(* Beckhoff Driver *)
	FBAxisToolLeftBeckhoff: FBHW_AXIS_SINGLE_BECKHOFF;
	FBAxisToolCenterBeckhoff: FBHW_AXIS_SINGLE_BECKHOFF;
	FBAxisToolRightBeckhoff: FBHW_AXIS_SINGLE_BECKHOFF;
	FBAxisToolFeederBeckhoff: FBHW_AXIS_SINGLE_BECKHOFF;
	FBAxisGrindFeederBeckhoff: FBHW_AXIS_SINGLE_BECKHOFF;
	FBLivevalueAxisToolLeftBeckhoff: FBHW_AXIS_LIVEVALUES_BECKHOFF;
	FBLivevalueAxisToolCenterBeckhoff: FBHW_AXIS_LIVEVALUES_BECKHOFF;
	FBLivevalueAxisToolRightBeckhoff: FBHW_AXIS_LIVEVALUES_BECKHOFF;
	FBLivevalueAxisToolFeederBeckhoff: FBHW_AXIS_LIVEVALUES_BECKHOFF;
	FBLivevalueAxisGrindFeederBeckhoff: FBHW_AXIS_LIVEVALUES_BECKHOFF;
	FBToolLeftMasterSlave:FBHW_AXIS_MULTI_BECKHOFF;
	FBToolCenterMasterSlave:FBHW_AXIS_MULTI_BECKHOFF;
	FBToolRightMasterSlave:FBHW_AXIS_MULTI_BECKHOFF;
	FBToolFeederMasterSlave:FBHW_AXIS_MULTI_BECKHOFF;
	FBCylToolTension : FBHW_CYL_ANALOGCYLINDER;
(*22.12.2009: KFS {    *)
	(*FBCalcToolTensionForce:FB_CALC_TOOLTENSION_FORCE;*)
	FBCalcToolTensionForce:FB_CALC_TOOLTENSION_FORCE_NEW;
	FBCylToolLeftActive:FBHW_CYL_STANDARD;
	FBCylToolRightActive:FBHW_CYL_STANDARD;
	FBCylToolCenterActive:FBHW_CYL_STANDARD;
	FBCylToolPrismaLeftActive:FBHW_CYL_STANDARD;
	FBCylToolPrismaRightActive:FBHW_CYL_STANDARD;
(*22.12.2009: KFS }   *)

(* Pointer auf Actuatoren *)
	ptrTAxisToolLeft:POINTER TO ST_AXIS;
	ptrTAxisToolCenter:POINTER TO ST_AXIS;
	ptrTAxisToolRight:POINTER TO ST_AXIS;
	ptrTAxisToolFeeder:POINTER TO ST_AXIS;
	ptrTAxisGrindFeeder:POINTER TO ST_AXIS;
	ptrTCylToolTension:POINTER TO ST_CYLINDER;
(*22.12.2009: KFS {    *)
	ptrTCylToolLeftActive:POINTER TO ST_CYLINDER;
	ptrTCylToolRightActive:POINTER TO ST_CYLINDER;
	ptrTCylToolCenterActive:POINTER TO ST_CYLINDER;
	ptrTCylToolPrismaLeftActive:POINTER TO ST_CYLINDER;
	ptrTCylToolPrismaRightActive:POINTER TO ST_CYLINDER;
	ptrTToolFeederWorkLength:POINTER TO ST_CYLINDER;
(*22.12.2009: KFS }   *)
	RisingEdgeHWConfig:R_TRIG;
	TONTickTime: TON;
	RisingEdgeSetError:R_TRIG;
	xHardwareConfigError: BOOL;
	xTmp: BOOL;
	xMicroRodActive: BOOL;
	xBeckhoffDriveActive: BOOL;
	xCkeckAcitveMovement: BOOL;

	axInputAxisToolLeftBeckhoff : ARRAY[1..8] OF BOOL;
	axInputAxisToolCenterBeckhoff : ARRAY[1..8] OF BOOL;
	axInputAxisToolRightBeckhoff : ARRAY[1..8] OF BOOL;
	axInputAxisToolFeederBeckhoff : ARRAY[1..8] OF BOOL;
	axInputAxisGrindFeederBeckhoff : ARRAY[1..8] OF BOOL;
	ii: INT;
	xFirstRead: BOOL;
	iStepResetHardware: INT;
	TONWaitReset: TON;
	rMaxWorkLength:REAL:=27;	 (* 0mm - 270mm = 0V - 10V  --> 270mm  --> Eingabe in cm! *)
	rMeasureWorkLengthCorrection:REAL:=0.4; (*Rundungs-Korrektur in cm*)
END_VAR
(****************************************************************************************************************************************************)
(***********                                            This Functionblock manage all the machine hardware                                                           ************)
(****************************************************************************************************************************************************)
(******************************************************************************************************************************************)
(****************************				              Activation Part                                                         *****************************)
(******************************************************************************************************************************************)
IF NOT(xFirstRead) THEN
	xFirstRead:=TRUE;
	TStation.THardware.TAxisToolLeft.T_RxPdoParameter.iControlWord:=6;
	TToolLeftRxPdoPara:=TStation.THardware.TAxisToolLeft.T_RxPdoParameter;
	TStation.THardware.TAxisToolCenter.T_RxPdoParameter.iControlWord:=6;
	TToolCenterRxPdoPara:=TStation.THardware.TAxisToolCenter.T_RxPdoParameter;
	TStation.THardware.TAxisToolRight.T_RxPdoParameter.iControlWord:=6;
	TToolRightRxPdoPara:=TStation.THardware.TAxisToolRight.T_RxPdoParameter;
	TStation.THardware.TAxisToolFeeder.T_RxPdoParameter.iControlWord:=6;
	TToolFeederRxPdoPara:=TStation.THardware.TAxisToolFeeder.T_RxPdoParameter;
	TStation.THardware.TAxisGrindFeeder.T_RxPdoParameter.iControlWord:=6;
	TGrindFeederRxPdoPara:=TStation.THardware.TAxisGrindFeeder.T_RxPdoParameter;
	(*06.12.2010 KFS:	{	*)
	T_Station.xOverwriteMaxToolLength:=FALSE;
	(*06.12.2010 KFS:	}	*)
END_IF;
IF TStation.TControl.xResetHardware THEN
	CASE iStepResetHardware OF
	1:	xResetControllerToolLeft:=TRUE;
		xResetControllerToolCenter:=TRUE;
		xResetControllerToolRight:=TRUE;
		xResetControllerToolFeeder:=TRUE;
		xResetControllerGrindFeeder:=TRUE;
		TONWaitReset(IN:=FALSE);
		iStepResetHardware:=iStepResetHardware + 1;
	2:	TONWaitReset(IN:=TRUE,PT:=T#100ms);
		IF TONWaitReset.Q THEN
			xResetControllerToolLeft:=FALSE;
			xResetControllerToolCenter:=FALSE;
			xResetControllerToolRight:=FALSE;
			xResetControllerToolFeeder:=FALSE;
			xResetControllerGrindFeeder:=FALSE;
			iStepResetHardware:=iStepResetHardware + 1;
		END_IF;
	3:	TStation.THardware.TAxisToolLeft.T_RxPdoParameter.iControlWord:=0;
		TToolLeftRxPdoPara:=TStation.THardware.TAxisToolLeft.T_RxPdoParameter;
		TStation.THardware.TAxisToolCenter.T_RxPdoParameter.iControlWord:=0;
		TToolCenterRxPdoPara:=TStation.THardware.TAxisToolCenter.T_RxPdoParameter;
		TStation.THardware.TAxisToolRight.T_RxPdoParameter.iControlWord:=0;
		TToolRightRxPdoPara:=TStation.THardware.TAxisToolRight.T_RxPdoParameter;
		TStation.THardware.TAxisToolFeeder.T_RxPdoParameter.iControlWord:=0;
		TToolFeederRxPdoPara:=TStation.THardware.TAxisToolFeeder.T_RxPdoParameter;
		TStation.THardware.TAxisGrindFeeder.T_RxPdoParameter.iControlWord:=0;
		TGrindFeederRxPdoPara:=TStation.THardware.TAxisGrindFeeder.T_RxPdoParameter;
		TONWaitReset(IN:=FALSE);
		iStepResetHardware:=iStepResetHardware + 1;
	4:	TONWaitReset(IN:=TRUE,PT:=T#100ms);
		IF TONWaitReset.Q THEN
			TStation.THardware.TAxisToolLeft.T_RxPdoParameter.iControlWord:=6;
			TToolLeftRxPdoPara:=TStation.THardware.TAxisToolLeft.T_RxPdoParameter;
			TStation.THardware.TAxisToolCenter.T_RxPdoParameter.iControlWord:=6;
			TToolCenterRxPdoPara:=TStation.THardware.TAxisToolCenter.T_RxPdoParameter;
			TStation.THardware.TAxisToolRight.T_RxPdoParameter.iControlWord:=6;
			TToolRightRxPdoPara:=TStation.THardware.TAxisToolRight.T_RxPdoParameter;
			TStation.THardware.TAxisToolFeeder.T_RxPdoParameter.iControlWord:=6;
			TToolFeederRxPdoPara:=TStation.THardware.TAxisToolFeeder.T_RxPdoParameter;
			TStation.THardware.TAxisGrindFeeder.T_RxPdoParameter.iControlWord:=6;
			TGrindFeederRxPdoPara:=TStation.THardware.TAxisGrindFeeder.T_RxPdoParameter;
			TONWaitReset(IN:=FALSE);
			iStepResetHardware:=1;
			TStation.TControl.xResetHardware:=FALSE;
		END_IF;
	END_CASE;
	RETURN;
ELSE
	iStepResetHardware:=1;
END_IF;
xActiveHWStation:=TStation.TControl.xActiveHardware;
RisingEdgeHWConfig(CLK:=xHardwareConfigError);
IF RisingEdgeHWConfig.Q THEN
	TStation.TControl.diErrorNr:=0;
	TStation.TControl.xError:=FALSE;
END_IF;
IF NOT(TStation.TControl.xActiveHardware) THEN
	TStation.TControl.xHWAxesActive:=TRUE;
	xHardwareConfigError:=FALSE;
	TONTickTime(IN:=FALSE);
	RisingEdgeSetError(CLK:=FALSE);
	TStation.TControl.xActiveMovement:=FALSE;
	RETURN;
ELSE
	(* Check Hardware Configuration *)
	IF TStation.TControl.xRdy THEN
		xTmp:=	(TStation.T_MachineConfig.iConfigMachineType <> iConfigMachineType) OR
				(TStation.T_MachineConfig.iConfigAxisType <> iConfigAxisType) OR
				(TStation.T_MachineConfig.iConfigVisuNavigation <> iConfigVisuNavigation) OR
				( (TStation.T_MachineConfig.rConfigMaxToolLength <> rConfigMaxToolLength) AND NOT(T_Station.xOverwriteMaxToolLength));
		IF xTmp THEN
			IF (TStation.T_MachineConfig.iConfigMachineType <> iConfigMachineType) THEN
				TStation.TControl.diErrorNr:=7001;	(* Error-->Config Machine Type changed *)
			END_IF;
			IF (TStation.T_MachineConfig.iConfigAxisType <> iConfigAxisType) THEN
				TStation.TControl.diErrorNr:=7002;	(* Error-->Config Axis Type changed *)
			END_IF;
			IF (TStation.T_MachineConfig.iConfigVisuNavigation <> iConfigVisuNavigation) THEN
				TStation.TControl.diErrorNr:=7003;	(* Error-->Config Visu Navigation changed *)
			END_IF;
			IF (TStation.T_MachineConfig.rConfigMaxToolLength <> rConfigMaxToolLength) THEN
				TStation.TControl.diErrorNr:=7004;	(* Error-->Config Max Tool Length changed *)
			END_IF;
			RisingEdgeSetError(CLK:=TRUE);
			IF RisingEdgeSetError.Q THEN
				TStation.TControl.xError:=TRUE;
			END_IF;
			xHardwareConfigError:=TRUE;
			TStation.TControl.xHardwareConfigError:=TRUE;
		END_IF;
	END_IF;
	IF xHardwareConfigError THEN
		TStation.TControl.xActiveMovement:=FALSE;
		RETURN;
	END_IF;
	IF NOT(TStation.TControl.xHardwareConfigError) THEN
		RisingEdgeSetError(CLK:=FALSE);
	END_IF;
	(* Zuweisung der Datenstrukturen der Aktuatoren als Pointer *)
	ptrTAxisToolLeft:=ADR(TStation.THardware.TAxisToolLeft);
	ptrTAxisToolCenter:=ADR(TStation.THardware.TAxisToolCenter);
	ptrTAxisToolRight:=ADR(TStation.THardware.TAxisToolRight);
	ptrTAxisToolFeeder:=ADR(TStation.THardware.TAxisToolFeeder);
	ptrTAxisGrindFeeder:=ADR(TStation.THardware.TAxisGrindFeeder);
	ptrTCylToolTension:=ADR(TStation.THardware.TCylToolTension);
(*22.12.2009: KFS {    *)
	ptrTCylToolLeftActive:=ADR(TStation.THardware.TCylToolLeftActive);
	ptrTCylToolRightActive:=ADR(TStation.THardware.TCylToolRightActive);
	ptrTCylToolCenterActive:=ADR(TStation.THardware.TCylToolCenterActive);
	ptrTCylToolPrismaLeftActive:=ADR(TStation.THardware.TCylToolPrismaLeftActive);
	ptrTCylToolPrismaRightActive:=ADR(TStation.THardware.TCylToolPrismaRightActive);
	ptrTToolFeederWorkLength:=ADR(TStation.THardware.TToolFeederWorkLength);
(*22.12.2009: KFS }   *)
	IF (iConfigMachineType = 2) THEN
		xMicroRodActive:=TRUE;
	ELSE
		xMicroRodActive:=FALSE;
	END_IF;
	IF (iConfigAxisType = 2) THEN
		xBeckhoffDriveActive:=TRUE;
	ELSE
		xBeckhoffDriveActive:=FALSE;
	END_IF;
END_IF;
(******************************************************************************************************************************************)
(****************************				         Check if Axis Active                                                    *****************************)
(******************************************************************************************************************************************)
xTmp:= ptrTAxisToolLeft^.T_CtrleSingle.xDone AND ptrTAxisToolRight^.T_CtrleSingle.xDone AND ptrTAxisToolFeeder^.T_CtrleSingle.xDone AND ptrTAxisGrindFeeder^.T_CtrleSingle.xDone;
xTmp:=xTmp AND ((ptrTAxisToolCenter^.T_CtrleSingle.xDone AND xMicroRodActive) OR NOT(xMicroRodActive));
IF xTmp THEN
	TStation.TControl.xHWAxesActive:=FALSE;
ELSE
	TStation.TControl.xHWAxesActive:=TRUE;
END_IF;
(******************************************************************************************************************************************)
(****************************	                        Check if Axis and Cylinder are Active                               *****************************)
(******************************************************************************************************************************************)
xCkeckAcitveMovement:=	(NOT(ptrTAxisToolLeft^.T_CtrleSingle.xDone) AND NOT(ptrTAxisToolLeft^.T_CtrleSingle.xErr)) OR
						(NOT(ptrTAxisToolRight^.T_CtrleSingle.xDone) AND NOT(ptrTAxisToolRight^.T_CtrleSingle.xErr)) OR
						(NOT(ptrTAxisToolFeeder^.T_CtrleSingle.xDone) AND NOT(ptrTAxisToolFeeder^.T_CtrleSingle.xErr)) OR
						(NOT(ptrTAxisGrindFeeder^.T_CtrleSingle.xDone) AND NOT(ptrTAxisGrindFeeder^.T_CtrleSingle.xErr)) OR
						(NOT(ptrTAxisToolCenter^.T_CtrleSingle.xDone) AND NOT(ptrTAxisToolCenter^.T_CtrleSingle.xErr) AND xMicroRodActive) OR
(*22.12.2009: KFS {    *)		(NOT(ptrTCylToolLeftActive^.T_CtrleCyl.xDone) AND NOT(ptrTCylToolLeftActive^.T_CtrleCyl.xErr) AND xMicroRodActive) OR
						(NOT(ptrTCylToolRightActive^.T_CtrleCyl.xDone) AND NOT(ptrTCylToolRightActive^.T_CtrleCyl.xErr) AND xMicroRodActive) OR
						(NOT(ptrTCylToolCenterActive^.T_CtrleCyl.xDone) AND NOT(ptrTCylToolCenterActive^.T_CtrleCyl.xErr) AND xMicroRodActive) OR
						(NOT(ptrTCylToolPrismaLeftActive^.T_CtrleCyl.xDone) AND NOT(ptrTCylToolPrismaLeftActive^.T_CtrleCyl.xErr) AND xMicroRodActive) OR
						(NOT(ptrTCylToolPrismaRightActive^.T_CtrleCyl.xDone) AND NOT(ptrTCylToolPrismaRightActive^.T_CtrleCyl.xErr) AND xMicroRodActive) OR	(*22.12.2009: KFS }   *)
						(NOT(ptrTCylToolTension^.T_CtrleCyl.xDone) AND NOT(ptrTCylToolTension^.T_CtrleCyl.xErr));
IF NOT(xCkeckAcitveMovement) THEN
	IF NOT(ptrTAxisToolLeft^.T_CtrleSingle.xNotMoving) AND ptrTAxisToolLeft^.T_CtrleSingle.xDone AND NOT(ptrTAxisToolLeft^.T_CtrleSingle.xErr) THEN
		xCkeckAcitveMovement:=TRUE;
	END_IF;
	IF NOT(ptrTAxisToolRight^.T_CtrleSingle.xNotMoving) AND ptrTAxisToolRight^.T_CtrleSingle.xDone AND NOT(ptrTAxisToolRight^.T_CtrleSingle.xErr) THEN
		xCkeckAcitveMovement:=TRUE;
	END_IF;
	IF NOT(ptrTAxisToolFeeder^.T_CtrleSingle.xNotMoving) AND ptrTAxisToolFeeder^.T_CtrleSingle.xDone AND NOT(ptrTAxisToolFeeder^.T_CtrleSingle.xErr) THEN
		xCkeckAcitveMovement:=TRUE;
	END_IF;
	IF NOT(ptrTAxisGrindFeeder^.T_CtrleSingle.xNotMoving) AND ptrTAxisGrindFeeder^.T_CtrleSingle.xDone AND NOT(ptrTAxisGrindFeeder^.T_CtrleSingle.xErr) THEN
		xCkeckAcitveMovement:=TRUE;
	END_IF;
	IF NOT(ptrTAxisToolCenter^.T_CtrleSingle.xNotMoving) AND ptrTAxisToolCenter^.T_CtrleSingle.xDone AND NOT(ptrTAxisToolCenter^.T_CtrleSingle.xErr) AND xMicroRodActive THEN
		xCkeckAcitveMovement:=TRUE;
	END_IF;
END_IF;
TStation.TControl.xActiveMovement:=xCkeckAcitveMovement;
IF NOT(xBeckhoffDriveActive) THEN
	(******************************************************************************************************************************************)
	(****************************				   Axis ToolLeft PDO Parameter                                      *****************************)
	(******************************************************************************************************************************************)
	TToolLeftRxPdoPara:=ptrTAxisToolLeft^.T_RxPdoParameter;
	ptrTAxisToolLeft^.T_TxPdoParameter:=TToolLeftTxPdoPara;
	(******************************************************************************************************************************************)
	(****************************				         Axis ToolLeft Live Values                                        *****************************)
	(******************************************************************************************************************************************)
	FBLivevalueAxisToolLeftEcostep(	iTypAxis:=1,
									rPrismaFactor:=0,
									xMicroRodActive:=xMicroRodActive,
									T_Axis:= ptrTAxisToolLeft^);
	(******************************************************************************************************************************************)
	(****************************				         Axis ToolLeft Motion                                                  *****************************)
	(******************************************************************************************************************************************)
	FBAxisToolLeftEcostep(	xCircuitPowerOn:= T_TwinSafeOut.QxContactor_K3 AND T_TwinSafeOut.QxContactor_K4,
							rPrismaFactor:=0,
							T_Axis:= ptrTAxisToolLeft^,
							T_HDD:= T_HDD);
	xResetControllerToolLeft:=FBAxisToolLeftEcostep.xResetController;
	xSetEnableAxisToolLeft:=FBAxisToolLeftEcostep.xSetEnableAxis;
	IF xMicroRodActive THEN
		(******************************************************************************************************************************************)
		(****************************		     	      Axis ToolCenter PDO Parameter                                      *****************************)
		(******************************************************************************************************************************************)
		TToolCenterRxPdoPara:=ptrTAxisToolCenter^.T_RxPdoParameter;
		ptrTAxisToolCenter^.T_TxPdoParameter:=TToolCenterTxPdoPara;
		(******************************************************************************************************************************************)
		(****************************				      Axis ToolCenter Live Values                                     *****************************)
		(******************************************************************************************************************************************)
		FBLivevalueAxisToolCenterEcostep(	iTypAxis:=2,
										rPrismaFactor:=0,
										xMicroRodActive:=xMicroRodActive,
										T_Axis:= ptrTAxisToolCenter^);
		(******************************************************************************************************************************************)
		(****************************				      Axis ToolCenter Motion                                               *****************************)
		(******************************************************************************************************************************************)
		FBAxisToolCenterEcostep(	xCircuitPowerOn:= T_TwinSafeOut.QxContactor_K3 AND T_TwinSafeOut.QxContactor_K4,
								rPrismaFactor:=0,
								T_Axis:= ptrTAxisToolCenter^,
								T_HDD:= T_HDD);
		xResetControllerToolCenter:=FBAxisToolCenterEcostep.xResetController;
		xSetEnableAxisToolCenter:=FBAxisToolCenterEcostep.xSetEnableAxis;
	ELSE
		xResetControllerToolCenter:=FALSE;
		xSetEnableAxisToolCenter:=FALSE;
	END_IF;
	(******************************************************************************************************************************************)
	(****************************			         Axis ToolRight PDO Parameter                                      *****************************)
	(******************************************************************************************************************************************)
	TToolRightRxPdoPara:=ptrTAxisToolRight^.T_RxPdoParameter;
	ptrTAxisToolRight^.T_TxPdoParameter:=TToolRightTxPdoPara;
	(******************************************************************************************************************************************)
	(****************************				        Axis ToolRight Live Values                                      *****************************)
	(******************************************************************************************************************************************)
	FBLivevalueAxisToolRightEcostep(	iTypAxis:=3,
									rPrismaFactor:=0,
									xMicroRodActive:=xMicroRodActive,
									T_Axis:= ptrTAxisToolRight^);
	(******************************************************************************************************************************************)
	(****************************				         Axis ToolRight Motion                                               *****************************)
	(******************************************************************************************************************************************)
	FBAxisToolRightEcostep(	xCircuitPowerOn:= T_TwinSafeOut.QxContactor_K3 AND T_TwinSafeOut.QxContactor_K4,
							rPrismaFactor:=0,
							T_Axis:= ptrTAxisToolRight^,
							T_HDD:= T_HDD);
	xResetControllerToolRight:=FBAxisToolRightEcostep.xResetController;
	xSetEnableAxisToolRight:=FBAxisToolRightEcostep.xSetEnableAxis;
	(******************************************************************************************************************************************)
	(****************************			      Axis ToolFeeder PDO Parameter                                    *****************************)
	(******************************************************************************************************************************************)
	TToolFeederRxPdoPara:=ptrTAxisToolFeeder^.T_RxPdoParameter;
	ptrTAxisToolFeeder^.T_TxPdoParameter:=TToolFeederTxPdoPara;
	(******************************************************************************************************************************************)
	(****************************				    Axis ToolFeeder Live Values                                     *****************************)
	(******************************************************************************************************************************************)
	FBLivevalueAxisToolFeederEcostep(	iTypAxis:=4,
										rPrismaFactor:=0,
										xMicroRodActive:=xMicroRodActive,
										T_Axis:= ptrTAxisToolFeeder^);
	(******************************************************************************************************************************************)
	(****************************				      Axis ToolFeeder Motion                                             *****************************)
	(******************************************************************************************************************************************)
	FBAxisToolFeederEcostep(	xCircuitPowerOn:= T_TwinSafeOut.QxContactor_K3 AND T_TwinSafeOut.QxContactor_K4,
								rPrismaFactor:=0,
								T_Axis:= ptrTAxisToolFeeder^,
								T_HDD:= T_HDD);
	xResetControllerToolFeeder:=FBAxisToolFeederEcostep.xResetController;
	xSetEnableAxisToolFeeder:=FBAxisToolFeederEcostep.xSetEnableAxis;
	(******************************************************************************************************************************************)
	(****************************			          Axis GrindFeeder PDO Parameter                               *****************************)
	(******************************************************************************************************************************************)
	TGrindFeederRxPdoPara:=ptrTAxisGrindFeeder^.T_RxPdoParameter;
	ptrTAxisGrindFeeder^.T_TxPdoParameter:=TGrindFeederTxPdoPara;
	(******************************************************************************************************************************************)
	(****************************				     Axis GrindFeeder Live Values                                   *****************************)
	(******************************************************************************************************************************************)
	FBLivevalueAxisGrindFeederEcostep(	iTypAxis:=5,
										rPrismaFactor:=rPrismaFactor,
										xMicroRodActive:=xMicroRodActive,
										T_Axis:= ptrTAxisGrindFeeder^);
	(******************************************************************************************************************************************)
	(****************************		           	      Axis GrindFeeder Motion                                            *****************************)
	(******************************************************************************************************************************************)
	FBAxisGrindFeederEcostep(	xCircuitPowerOn:= T_TwinSafeOut.QxContactor_K3 AND T_TwinSafeOut.QxContactor_K4,
								rPrismaFactor:=rPrismaFactor,
								T_Axis:= ptrTAxisGrindFeeder^,
								T_HDD:= T_HDD);
	xResetControllerGrindFeeder:=FBAxisGrindFeederEcostep.xResetController;
	xSetEnableAxisGrindFeeder:=FBAxisGrindFeederEcostep.xSetEnableAxis;
END_IF;
IF xBeckhoffDriveActive THEN
	(******************************************************************************************************************************************)
	(****************************				         Axis ToolLeft Live Values                                        *****************************)
	(******************************************************************************************************************************************)
	FOR ii:=1 TO 8 DO
		axInputAxisToolLeftBeckhoff[ii]:=axInputAxisBeckhoff[1,ii];
	END_FOR
	FBLivevalueAxisToolLeftBeckhoff(	uiActualTorque:=auiActualAxisTorqueBeckhoff[1],
									arxDigitalInput:=axInputAxisToolLeftBeckhoff,
									T_AXIS:=ptrTAxisToolLeft^,
									T_AXISRefIn:=stToolLeftRefIn);

	(******************************************************************************************************************************************)
	(****************************				         Axis ToolLeft Motion                                                  *****************************)
	(******************************************************************************************************************************************)
	FBAxisToolLeftBeckhoff(	xHWLimitPos:= FALSE,
							xHWLimitNeg:= FALSE,
							xRefHoming:= FALSE,
							T_Axis:= ptrTAxisToolLeft^,
							T_AxisRefIn:= stToolLeftRefIn,
							T_AxisRefOut:= stToolLeftRefOut,
							T_HDD:= T_HDD);

	(******************************************************************************************************************************************)
	(****************************				            Axis ToolLeft Mulit                                                    *****************************)
	(******************************************************************************************************************************************)
	IF xMicroRodActive THEN
		FBToolLeftMasterSlave(	T_AxisMaster:=ptrTAxisToolLeft^ ,
								T_AxisSlave:= ptrTAxisToolCenter^,
								T_AxisMasterRefIn:= stToolLeftRefIn,
								T_AxisSlaveRefIn:= stToolCenterRefIn);
	ELSE
		FBToolLeftMasterSlave(	T_AxisMaster:=ptrTAxisToolLeft^ ,
								T_AxisSlave:= ptrTAxisToolRight^,
								T_AxisMasterRefIn:= stToolLeftRefIn,
								T_AxisSlaveRefIn:= stToolRightRefIn);
	END_IF;

	IF xMicroRodActive THEN
		(******************************************************************************************************************************************)
		(****************************				      Axis ToolCenter Live Values                                     *****************************)
		(******************************************************************************************************************************************)
		FOR ii:=1 TO 8 DO
			axInputAxisToolCenterBeckhoff[ii]:=axInputAxisBeckhoff[2,ii];
		END_FOR
		FBLivevalueAxisToolCenterBeckhoff(	uiActualTorque:=auiActualAxisTorqueBeckhoff[2],
										arxDigitalInput:=axInputAxisToolCenterBeckhoff,
										T_AXIS:=ptrTAxisToolCenter^,
										T_AXISRefIn:=stToolCenterRefIn);

		(******************************************************************************************************************************************)
		(****************************				      Axis ToolCenter Motion                                               *****************************)
		(******************************************************************************************************************************************)
		FBAxisToolCenterBeckhoff(	xHWLimitPos:= FALSE,
								xHWLimitNeg:= FALSE,
								xRefHoming:= FALSE,
								T_Axis:= ptrTAxisToolCenter^,
								T_AxisRefIn:= stToolCenterRefIn,
								T_AxisRefOut:= stToolCenterRefOut,
								T_HDD:= T_HDD);

		(******************************************************************************************************************************************)
		(****************************				        Axis ToolCenter Mulit                                                 *****************************)
		(******************************************************************************************************************************************)
		FBToolCenterMasterSlave(	T_AxisMaster:=ptrTAxisToolCenter^ ,
								T_AxisSlave:= ptrTAxisToolRight^,
								T_AxisMasterRefIn:= stToolCenterRefIn,
								T_AxisSlaveRefIn:= stToolRightRefIn);
	END_IF;

	(******************************************************************************************************************************************)
	(****************************				        Axis ToolRight Live Values                                      *****************************)
	(******************************************************************************************************************************************)
	FOR ii:=1 TO 8 DO
		axInputAxisToolRightBeckhoff[ii]:=axInputAxisBeckhoff[3,ii];
	END_FOR
	FBLivevalueAxisToolRightBeckhoff(	uiActualTorque:=auiActualAxisTorqueBeckhoff[3],
									arxDigitalInput:=axInputAxisToolRightBeckhoff,
									T_AXIS:=ptrTAxisToolRight^,
									T_AXISRefIn:=stToolRightRefIn);

	(******************************************************************************************************************************************)
	(****************************				         Axis ToolRight Motion                                               *****************************)
	(******************************************************************************************************************************************)
	FBAxisToolRightBeckhoff(	xHWLimitPos:= FALSE,
							xHWLimitNeg:= FALSE,
							xRefHoming:= FALSE,
							T_Axis:= ptrTAxisToolRight^,
							T_AxisRefIn:= stToolRightRefIn,
							T_AxisRefOut:= stToolRightRefOut,
							T_HDD:= T_HDD);

	(******************************************************************************************************************************************)
	(****************************				            Axis ToolRight Mulit                                                *****************************)
	(******************************************************************************************************************************************)
	FBToolRightMasterSlave(	T_AxisMaster:=ptrTAxisToolRight^ ,
							T_AxisSlave:= ptrTAxisToolFeeder^,
							T_AxisMasterRefIn:= stToolRightRefIn,
							T_AxisSlaveRefIn:= stToolFeederRefIn);

	(******************************************************************************************************************************************)
	(****************************				    Axis ToolFeeder Live Values                                     *****************************)
	(******************************************************************************************************************************************)
	FOR ii:=1 TO 8 DO
		axInputAxisToolFeederBeckhoff[ii]:=axInputAxisBeckhoff[4,ii];
	END_FOR
	FBLivevalueAxisToolFeederBeckhoff(	uiActualTorque:=auiActualAxisTorqueBeckhoff[4],
										arxDigitalInput:=axInputAxisToolFeederBeckhoff,
										T_AXIS:=ptrTAxisToolFeeder^,
										T_AXISRefIn:=stToolFeederRefIn);

	(******************************************************************************************************************************************)
	(****************************				      Axis ToolFeeder Motion                                             *****************************)
	(******************************************************************************************************************************************)
	FBAxisToolFeederBeckhoff(	xHWLimitPos:= FALSE,
								xHWLimitNeg:= FALSE,
								xRefHoming:= FALSE,
								T_Axis:= ptrTAxisToolFeeder^,
								T_AxisRefIn:= stToolFeederRefIn,
								T_AxisRefOut:= stToolFeederRefOut,
								T_HDD:= T_HDD);

	(******************************************************************************************************************************************)
	(****************************				            Axis ToolFeeder Mulit                                            *****************************)
	(******************************************************************************************************************************************)
	FBToolFeederMasterSlave(T_AxisMaster:=ptrTAxisToolFeeder^ ,
							T_AxisSlave:= ptrTAxisGrindFeeder^,
							T_AxisMasterRefIn:= stToolFeederRefIn,
							T_AxisSlaveRefIn:= stGrindFeederRefIn);

	(******************************************************************************************************************************************)
	(****************************				     Axis GrindFeeder Live Values                                   *****************************)
	(******************************************************************************************************************************************)
	FOR ii:=1 TO 8 DO
		axInputAxisGrindFeederBeckhoff[ii]:=axInputAxisBeckhoff[5,ii];
	END_FOR
	FBLivevalueAxisGrindFeederBeckhoff(	uiActualTorque:=auiActualAxisTorqueBeckhoff[5],
										arxDigitalInput:=axInputAxisGrindFeederBeckhoff,
										T_AXIS:=ptrTAxisGrindFeeder^,
										T_AXISRefIn:=stGrindFeederRefIn);

	(******************************************************************************************************************************************)
	(****************************		           	      Axis GrindFeeder Motion                                            *****************************)
	(******************************************************************************************************************************************)
	FBAxisGrindFeederBeckhoff(	xHWLimitPos:= FALSE,
								xHWLimitNeg:= FALSE,
								xRefHoming:= FALSE,
								T_Axis:= ptrTAxisGrindFeeder^,
								T_AxisRefIn:= stGrindFeederRefIn,
								T_AxisRefOut:= stGrindFeederRefOut,
								T_HDD:= T_HDD);

	(******************************************************************************************************************************************)
	(****************************				           Axis GrindFeeder Mulit                                            *****************************)
	(******************************************************************************************************************************************)
	(* No Slave Axis for Axis GrindFeeder *)
END_IF;

(******************************************************************************************************************************************)
(****************************		                       Cylinder für  ToolTension                                             *****************************)
(******************************************************************************************************************************************)
FBCalcToolTensionForce(	rForcePistonIn:= ptrTCylToolTension^.T_CtrleCyl.T_AnalogCylinder.rForceIn,
						rPistonDiameterD1:= T_ParamToolTensionSystem.rPistonDiameterTT,
						rPistonDiameterD2:= T_ParamToolTensionSystem.rPistonDiameterTT2,
						rMaxAirpressure:= T_ParamToolTensionSystem.rAirPressureTT,
						rFactorForce:= T_ParamToolTensionSystem.rFactorForce);
T_ParamToolTensionSystem.rMaxForceTT:=FBCalcToolTensionForce.rSetMaxForce;
ptrTCylToolTension^.T_CtrleCyl.T_AnalogCylinder.iAnalogIN:=FBCalcToolTensionForce.iAnalogOutput;
ptrTCylToolTension^.T_CtrleCyl.T_AnalogCylinder.rForceOut:=FBCalcToolTensionForce.rForcePistonOut;
FBCylToolTension(	xCtrlePosOn:=xSensorToolTension,
					xCtrlePosOff:=FALSE,
					iAnalogIn:= ptrTCylToolTension^.T_CtrleCyl.T_AnalogCylinder.iAnalogIN,
					T_Cylinder:= ptrTCylToolTension^);
iCylOutAnaToolTension:=FBCylToolTension.iAnalogOut;
ptrTCylToolTension^.T_CtrleCyl.T_AnalogCylinder.iAnalogOut:=FBCylToolTension.iAnalogOut;
xCylOutToolTension:=FBCylToolTension.xCylinder;
IF xMicroRodActive THEN
	(* control lamp button for the Cylinder ToolTension *)
	xCtrlLampToolTensionButton:=FBCylToolTension.xCylinder;
END_IF
(******************************************************************************************************************************************)
IF xMicroRodActive THEN
	(******************************************************************************************************************************************)
	(****************************		                       Cylinder für  ToolLeftActive                                          *****************************)
	(******************************************************************************************************************************************)
	FBCylToolLeftActive(		xCtrlePosOn:= FALSE,
							xCtrlePosOff:= FALSE,
							T_Cylinder:= ptrTCylToolLeftActive^);
	xCylOutToolLeftActive:= FBCylToolLeftActive.xCylinder;
	(* control lamp button for the Cylinder ToolLeft *)
	xCtrlLampToolLeftButton:= FBCylToolLeftActive.xCylinder;
	(******************************************************************************************************************************************)
	(****************************		                       Cylinder für  ToolRightActive                                       *****************************)
	(******************************************************************************************************************************************)
	FBCylToolRightActive(		xCtrlePosOn:= FALSE,
							xCtrlePosOff:= FALSE,
							T_Cylinder:= ptrTCylToolRightActive^);
	xCylOutToolRightActive:= FBCylToolRightActive.xCylinder;
	(* control lamp button for the Cylinder ToolRight*)
	xCtrlLampToolRightButton:= FBCylToolRightActive.xCylinder;
	(******************************************************************************************************************************************)
	(****************************		                       Cylinder für  ToolCenterActive                                       *****************************)
	(******************************************************************************************************************************************)
	FBCylToolCenterActive(	xCtrlePosOn:= FALSE,
							xCtrlePosOff:= FALSE,
							T_Cylinder:= ptrTCylToolCenterActive^);
	xCylOutToolCenterActive:= FBCylToolCenterActive.xCylinder;
	(* control lamp button for the Cylinder ToolCenter *)
	xCtrlLampToolCenterButton:= FBCylToolCenterActive.xCylinder;
	(******************************************************************************************************************************************)
	(****************************		                       Cylinder für  ToolPrismaLeftActive                            *****************************)
	(******************************************************************************************************************************************)
	FBCylToolPrismaLeftActive(	xCtrlePosOn:= FALSE,
								xCtrlePosOff:= FALSE,
								T_Cylinder:= ptrTCylToolPrismaLeftActive^);
	xCylOutToolPrismaLeftActive:= FBCylToolPrismaLeftActive.xCylinder;
	(* control lamp button for the Cylinder ToolPrismaLeft *)
	xCtrlLampToolPrismaLeftButton:= FBCylToolPrismaLeftActive.xCylinder;
	(******************************************************************************************************************************************)
	(****************************		                       Cylinder für  ToolPrismaRightActive                         *****************************)
	(******************************************************************************************************************************************)
	FBCylToolPrismaRightActive(	xCtrlePosOn:= FALSE,
								xCtrlePosOff:= FALSE,
								T_Cylinder:= ptrTCylToolPrismaRightActive^);
	xCylOutToolPrismaRightActive:= FBCylToolPrismaRightActive.xCylinder;
	(* control lamp button for the Cylinder ToolPrismaRight *)
	xCtrlLampToolPrismaRightButton:= FBCylToolPrismaRightActive.xCylinder;
	(************************************************************************************************************************************************************)
	(****************************		              Calculation for the ToolFeederWorkLength                    ***********************************************)
	(************************************************************************************************************************************************************)
	ptrTToolFeederWorkLength^.T_CtrleCyl.T_Analog.rLengthIn:=((rMaxWorkLength/32767) * INT_TO_REAL(iAToolFeederWorkLength)) - rMeasureWorkLengthCorrection;
	(************************************************************************************************************************************************************)
END_IF;
(******************************************************************************************************************************************)
(****************************		                              Reset Control Flags                                                *****************************)
(******************************************************************************************************************************************)
ptrTAxisToolLeft^.T_CtrleSingle.xExecute:=FALSE;
ptrTAxisToolLeft^.T_CtrleSingle.xReset:=FALSE;
ptrTAxisToolCenter^.T_CtrleSingle.xExecute:=FALSE;
ptrTAxisToolCenter^.T_CtrleSingle.xReset:=FALSE;
ptrTAxisToolRight^.T_CtrleSingle.xExecute:=FALSE;
ptrTAxisToolRight^.T_CtrleSingle.xReset:=FALSE;
ptrTAxisToolFeeder^.T_CtrleSingle.xExecute:=FALSE;
ptrTAxisToolFeeder^.T_CtrleSingle.xReset:=FALSE;
ptrTAxisGrindFeeder^.T_CtrleSingle.xExecute:=FALSE;
ptrTAxisGrindFeeder^.T_CtrleSingle.xReset:=FALSE;
ptrTCylToolTension^.T_CtrleCyl.xReset:=FALSE;
ptrTCylToolTension^.T_CtrleCyl.xExecute:=FALSE;
ptrTCylToolLeftActive^.T_CtrleCyl.xReset:=FALSE;
ptrTCylToolLeftActive^.T_CtrleCyl.xExecute:=FALSE;
ptrTCylToolRightActive^.T_CtrleCyl.xReset:=FALSE;
ptrTCylToolRightActive^.T_CtrleCyl.xExecute:=FALSE;
ptrTCylToolCenterActive^.T_CtrleCyl.xReset:=FALSE;
ptrTCylToolCenterActive^.T_CtrleCyl.xExecute:=FALSE;
ptrTCylToolPrismaLeftActive^.T_CtrleCyl.xReset:=FALSE;
ptrTCylToolPrismaLeftActive^.T_CtrleCyl.xExecute:=FALSE;
ptrTCylToolPrismaRightActive^.T_CtrleCyl.xReset:=FALSE;
ptrTCylToolPrismaRightActive^.T_CtrleCyl.xExecute:=FALSE;
ptrTToolFeederWorkLength^.T_CtrleCyl.xReset:=FALSE;
ptrTToolFeederWorkLength^.T_CtrleCyl.xExecute:=FALSE;
END_FUNCTION_BLOCK

(* POU FB_HARDWARE/FBHW_AXIS_SINGLE_ECOSTEP, ST *)
FUNCTION_BLOCK FBHW_AXIS_SINGLE_ECOSTEP
VAR_INPUT
	xCircuitPowerOn:BOOL;
	rPrismaFactor:REAL;
END_VAR
VAR_OUTPUT
	xResetController:BOOL;
	xSetEnableAxis:BOOL;
END_VAR
VAR_IN_OUT
	T_Axis:ST_AXIS;
	T_HDD:ST_HDD;
END_VAR
VAR
	siOpMode:SINT;
	uiStatusWord:UINT;
	FBConvertPdoMapping:FB_CONVERT_PDOMAPPING;
	FBConvertAxisParameter:FB_CONVERT_AXISPARAMETER;
(*fbDefaultAxisPara:FBDefaultAxisValue; *)
	FBGetObjectSDO:FB_GetObject;
	FBSetObjectSDO:FB_SetObject;
(* timer *)
	TimerFileLocked:TON;
(* trigger *)
	RisingEdgeStop:R_TRIG;
	RisingEdgeResetFB:R_TRIG;
	RisingEdgeExecute:R_TRIG;
	RisingEdgePowerOn:R_TRIG;
	RisingEdgePowerOff:R_TRIG;
(* variable *)
	xConfirmResetFB:BOOL;
	xReadFault:BOOL;
	xResetAxis:BOOL;
	xPowerOn:BOOL;
	xPowerOff:BOOL;
	xStop:BOOL;
	xMoveVel:BOOL;
	xMoveAbs:BOOL;
	xMoveRel:BOOL;
	xHoming:BOOL;
	xCalcAngleRefIndex:BOOL;
	xSetPosition:BOOL;
	xNewVelocity:BOOL;
	xNewPosition:BOOL;
	xSetOperationMode:BOOL;
	xReadFile:BOOL;
	xWriteFile:BOOL;
	xSendAxisParameter:BOOL;
	xRestoreAxisPower:BOOL;
	xConfirmRequest:BOOL;
	xDriveTorqueIn:BOOL;
	xDriveTorqueOut:BOOL;
	xSetTorqueValue:BOOL;
	iStepSendPara:INT:=0;
	iPtrAxisParameter:INT:=0;
	iStepResetFB:INT;
	iStepFile:INT;
	iStepDriveTorque:INT;
	xConfirmDone:BOOL;
	xConfirmErr:BOOL;
	udiConfirmErrorID:UDINT;
(* temporary variable *)
	i:INT;
	sTmp:STRING(255);
	sDeleteDataAxis: ARRAY[1..csiMaxAxisFileObj] OF STRING(120);
	sDeleteDataHDD: ARRAY[1..csiMaxFileLine] OF STRING(255);
	xSendPDOMappingPara: BOOL;
	xReadFilePDOMappingPara: BOOL;
	SetObjectSDO: BOOL;
	GetObjectSDO: BOOL;
	udiIdxGroup: UDINT;
	udiIndexOffset: UDINT;
	udiLength: UDINT;
	lrReal: LREAL;
	iStepMoveVel: INT;
	iStepStop: INT;
	iStepPowerOn: INT;
	iStepPowerOff: INT;
	iStepMovePos: INT;
	iStepResetAxis: INT;
	iStepSetPosition: INT;
	xMasterSlave: BOOL;
	iStepMasterSlave: INT;
	iStepHoming: INT;
	iStepReadFile: INT;
	lrSettledControlword:LREAL;
	xReadError: BOOL;
	xBlockReadError: BOOL;
	WaitSwitchReady: TON;
	iStepCalcAngleRefIndex: INT;
	xSaveParaEcoDrive: BOOL;
	iStepSaveParaEcoDrive: INT;
	xGetSoftwareVersion: BOOL;
	iStepGetSoftwareVersion: INT;
	sTmpDateCode: STRING(16);
	sCopyDateCode: STRING(16);
	xADSErrorActive: BOOL;
	udiADSErrorID: UDINT;
	xFBErrorActive: BOOL;
	udiFBErrorID: UDINT;
	TimerFunctionTimeOut: TON;
	tTimeOutFunction: TIME;
	lrCapturePosition: LREAL;
	xTmp: BOOL;
	xBlockFBFunction: BOOL;
	iStepBlockFunction: INT;
	xFirstRead: BOOL;
	xNotMoving: BOOL;
	sTmp1: STRING;
	xSetSWLimitSwitch: BOOL;
	iStepSetSWLimitSwitch: INT;
	xResetSWLimitSwitch: BOOL;
	iStepResetSWLimitSwitch: INT;
	xTmp1: BOOL;
	xTmp2: BOOL;
	lrForceSpeed: LREAL;
	TONWaitSetValue: TON;
END_VAR
(****************************************************************************************************************************************************)
(***********                                               This Functionblock is the driver for the EcoStep Axis                                                           ************)
(****************************************************************************************************************************************************)
(* First read *)
	IF NOT(xFirstRead) THEN
		xFirstRead:=TRUE;
		TimerFunctionTimeOut(IN:=FALSE);
		tTimeOutFunction:=T#999999s;
	END_IF;
(* reset block function *)
	RisingEdgeResetFB(CLK:=T_Axis.T_CtrleSingle.xReset);
	IF RisingEdgeResetFB.Q THEN
	(* Init. block function *)
		(* Init. variable *)
		IF T_Axis.T_CtrleSingle.xErr THEN
			xSetEnableAxis:=FALSE;
		END_IF;
		xNotMoving:=TRUE;
		xReadFault:=FALSE;
		xNewVelocity:=FALSE;
		xNewPosition:=FALSE;
		xSetOperationMode:=FALSE;
		xWriteFile:=FALSE;
		xRestoreAxisPower:=FALSE;
		xConfirmRequest:=FALSE;
		xDriveTorqueIn:=FALSE;
		xDriveTorqueOut:=FALSE;
		xSetTorqueValue:=FALSE;
		xResetAxis:=xReadFile:=xPowerOn:=xPowerOff:=xStop:=	xMoveVel:=xMoveAbs:=xMoveRel:=xHoming:=	xSetPosition:=xCalcAngleRefIndex:=FALSE;
		xSendAxisParameter:=xReadFilePDOMappingPara:=xSendPDOMappingPara:=xMasterSlave:=xSaveParaEcoDrive:=xGetSoftwareVersion:=FALSE;
		xSetSWLimitSwitch:=xResetSWLimitSwitch:=FALSE;
		xBlockFBFunction:=FALSE;
		iStepResetFB:=0;
		iStepFile:=0;
		iStepDriveTorque:=0;
		xConfirmDone:=FALSE;
		xConfirmErr:=FALSE;
		udiConfirmErrorID:=0;
		TimerFunctionTimeOut(IN:=FALSE);
		tTimeOutFunction:=T#999999s;
		(* int. structure *)
		T_Axis.T_CtrleSingle.dwOverride:=100;
		T_Axis.T_CtrleSingle.iFunction:=0;
		T_Axis.T_CtrleSingle.xDone:=FALSE;
		T_Axis.T_CtrleSingle.xErr:=FALSE;
		T_Axis.T_CtrleSingle.udiErrorID:=0;
		T_Axis.T_CtrleSingle.xPower:=FALSE;
		T_Axis.T_CtrleSingle.xReady:=FALSE;
		T_Axis.T_CtrleSingle.xNotMoving:=FALSE;
		T_Axis.T_CtrleSingle.xRef:=FALSE;
		T_Axis.T_CtrleSingle.xSlave:=FALSE;
		T_Axis.T_CtrleSingle.xBusyNewPosAndVel:=FALSE;
		T_Axis.T_CtrleSingle.xDriveTorque:=FALSE;
		(* set flag done *)
		xConfirmResetFB:=TRUE;
		(* exit function bloc *)
		RETURN;
	ELSE
		IF xConfirmResetFB THEN
		(* confirm reset FB *)
			T_Axis.T_CtrleSingle.xDone:=TRUE;
			T_Axis.T_CtrleSingle.xErr:=FALSE;
			T_Axis.T_CtrleSingle.udiErrorID:=0;
			(* reset variable *)
			xConfirmResetFB:=FALSE;
		END_IF
	END_IF

(* return axis state *)
	siOpMode:=T_Axis.T_TxPdoParameter.siOperationModesDisplay;
	uiStatusWord:=T_Axis.T_TxPdoParameter.uiStatusWord;
	T_Axis.T_CtrleSingle.xReady:=		TRUE;
	T_Axis.T_CtrleSingle.xPower:=		GETBIT32(uiStatusWord,0) AND GETBIT32(uiStatusWord,1) AND GETBIT32(uiStatusWord,2) AND NOT(GETBIT32(uiStatusWord,3)) AND
									GETBIT32(uiStatusWord,4) AND GETBIT32(uiStatusWord,5) AND GETBIT32(uiStatusWord,14) AND xSetEnableAxis AND xCircuitPowerOn;
	T_Axis.T_CtrleSingle.xRef:=			GETBIT32(uiStatusWord,15);
	T_Axis.T_CtrleSingle.xSlave:=		(siOpMode = -4);
	T_Axis.T_CtrleSingle.xNotMoving:=	xNotMoving;

(* check HW Axis Error and read it *)
	IF ((UINT_TO_WORD(uiStatusWord) AND 16#8) = 16#8) AND NOT(xReadError) THEN
		IF NOT(GetObjectSDO) THEN
			udiIdxGroup:=16#2600;	(* Error Object *)
			udiIndexOffset:=16#2;
			udiLength:=16#4;
			GetObjectSDO:=TRUE;
			xReadError:=TRUE;
			xResetAxis:=xReadFile:=xPowerOn:=xPowerOff:=xStop:=	xMoveVel:=xMoveAbs:=xMoveRel:=xHoming:=	xSetPosition:=xCalcAngleRefIndex:=FALSE;
			xSendAxisParameter:=xReadFilePDOMappingPara:=xSendPDOMappingPara:=xMasterSlave:=xSaveParaEcoDrive:=xGetSoftwareVersion:=FALSE;
			xSetSWLimitSwitch:=xResetSWLimitSwitch:=FALSE;
		END_IF;
	ELSE
		IF ((UINT_TO_WORD(uiStatusWord) AND 16#8) = 16#8) AND NOT(GetObjectSDO) AND NOT(xBlockReadError) AND xReadError THEN
			T_Axis.T_CtrleSingle.udiErrorID:=FCT_GET_AXIS_ERROR(LREAL_TO_DWORD(lrReal));
			T_Axis.T_CtrleSingle.xDone:=FALSE;
			T_Axis.T_CtrleSingle.xErr:=TRUE;
			xBlockReadError:=TRUE;
			xNotMoving:=TRUE;
		END_IF;
		IF ((UINT_TO_WORD(uiStatusWord) AND 16#8) = 16#0) THEN
			xReadError:=FALSE;
			xBlockReadError:=FALSE;
		END_IF;
	END_IF;

(* check ADS communication Error *)
	IF xADSErrorActive THEN
		xResetAxis:=xReadFile:=xPowerOn:=xPowerOff:=xStop:=	xMoveVel:=xMoveAbs:=xMoveRel:=xHoming:=	xSetPosition:=xCalcAngleRefIndex:=FALSE;
		xSendAxisParameter:=xReadFilePDOMappingPara:=xSendPDOMappingPara:=xMasterSlave:=xSaveParaEcoDrive:=xGetSoftwareVersion:=FALSE;
		xSetSWLimitSwitch:=xResetSWLimitSwitch:=FALSE;
		(* T_Axis.T_CtrleSingle.udiErrorID:=udiADSErrorID + 16#10000000;	(* With the Value 16#10000000 it can detect an error from the ADS communication *) *)
		T_Axis.T_CtrleSingle.udiErrorID:=16#F214;
		T_Axis.T_CtrleSingle.xErr:=TRUE;
		T_Axis.T_CtrleSingle.xDone:=FALSE;
		xADSErrorActive:=FALSE;
		FBSetObjectSDO(Write:=FALSE);
		FBGetObjectSDO(Read:=FALSE);
		xNotMoving:=TRUE;
	END_IF;

(* check FB Error *)
	IF xFBErrorActive THEN
		xResetAxis:=xReadFile:=xPowerOn:=xPowerOff:=xStop:=	xMoveVel:=xMoveAbs:=xMoveRel:=xHoming:=	xSetPosition:=xCalcAngleRefIndex:=FALSE;
		xSendAxisParameter:=xReadFilePDOMappingPara:=xSendPDOMappingPara:=xMasterSlave:=xSaveParaEcoDrive:=xGetSoftwareVersion:=FALSE;
		xSetSWLimitSwitch:=xResetSWLimitSwitch:=FALSE;
		T_Axis.T_CtrleSingle.xDone:=FALSE;
		T_Axis.T_CtrleSingle.xErr:=TRUE;
		T_Axis.T_CtrleSingle.udiErrorID:=udiFBErrorID;	(* FB Error can detect with prefix 16#2... *)
		xFBErrorActive:=FALSE;
		xNotMoving:=TRUE;
		xResetController:=FALSE;
	END_IF;
	IF TimerFunctionTimeOut.Q AND NOT(T_Axis.T_CtrleSingle.xDone) AND NOT(T_Axis.T_CtrleSingle.xErr) THEN
		xResetAxis:=xReadFile:=xPowerOn:=xPowerOff:=xStop:=	xMoveVel:=xMoveAbs:=xMoveRel:=xHoming:=	xSetPosition:=xCalcAngleRefIndex:=FALSE;
		xSendAxisParameter:=xReadFilePDOMappingPara:=xSendPDOMappingPara:=xMasterSlave:=xSaveParaEcoDrive:=xGetSoftwareVersion:=FALSE;
		xSetSWLimitSwitch:=xResetSWLimitSwitch:=FALSE;
		T_Axis.T_CtrleSingle.xDone:=FALSE;
		T_Axis.T_CtrleSingle.xErr:=TRUE;
		T_Axis.T_CtrleSingle.udiErrorID:=16#F206;	(* Axis Function time out error *)
		xNotMoving:=TRUE;
		xResetController:=FALSE;
	END_IF;

(* check while movement the SW and HW limitswitch *)
	xTmp:= T_Axis.T_CtrleSingle.xHWLimitNeg OR T_Axis.T_CtrleSingle.xHWLimitPos OR T_Axis.T_CtrleSingle.xSWLimitNeg OR T_Axis.T_CtrleSingle.xSWLimitPos;

	xTmp1:= NOT(xMoveAbs) AND NOT(xMoveRel) AND NOT(xMoveVel) AND NOT(T_Axis.T_CtrleSingle.xNotMoving) AND NOT(T_Axis.T_CtrleSingle.xErr);

	xTmp1:= xTmp1 AND ( (T_Axis.T_CtrleSingle.lrSWNegLimitSwitch <> 0.0) OR (T_Axis.T_CtrleSingle.lrSWPosLimitSwitch <> 0.0) );

	IF xTmp1 THEN
		IF ( (T_Axis.T_LiveValue.lrActualPosition < T_Axis.T_CtrleSingle.lrSWNegLimitSwitch) OR
		      (T_Axis.T_LiveValue.lrActualPosition > T_Axis.T_CtrleSingle.lrSWPosLimitSwitch)      ) THEN
			xTmp2:=TRUE;
		ELSE
			xTmp2:=FALSE;
		END_IF;
	ELSE
		xTmp2:=FALSE;
	END_IF;

	IF ( xTmp OR xTmp2 OR xBlockFBFunction ) AND NOT(T_Axis.T_CtrleSingle.xErr) THEN
		IF ( xMoveAbs OR xMoveRel OR xMoveVel OR xTmp2 OR NOT(T_Axis.T_CtrleSingle.xNotMoving) ) AND NOT(xStop) AND NOT(xBlockFBFunction) THEN
			xBlockFBFunction:=TRUE;
			IF xMoveAbs THEN
				IF ( (T_Axis.T_CtrleSingle.lrPosition >= T_Axis.T_CtrleSingle.lrSWNegLimitSwitch) AND (T_Axis.T_CtrleSingle.lrPosition <= T_Axis.T_CtrleSingle.lrSWPosLimitSwitch)) THEN
					xBlockFBFunction:=FALSE;
				END_IF;
			      IF T_Axis.T_LiveValue.lrActualPosition - T_Axis.T_CtrleSingle.lrPosition  < 0 AND T_Axis.T_CtrleSingle.xHWLimitNeg THEN
					xBlockFBFunction:=FALSE;
				END_IF
				IF  T_Axis.T_LiveValue.lrActualPosition - T_Axis.T_CtrleSingle.lrPosition > 0 AND T_Axis.T_CtrleSingle.xHWLimitPos THEN
					xBlockFBFunction:=FALSE;
				END_IF;
			END_IF;
			IF xMoveRel THEN
				IF ( (T_Axis.T_LiveValue.lrActualPosition + T_Axis.T_CtrleSingle.lrDistance) >= T_Axis.T_CtrleSingle.lrSWNegLimitSwitch ) AND
				    ( (T_Axis.T_LiveValue.lrActualPosition + T_Axis.T_CtrleSingle.lrDistance) <= T_Axis.T_CtrleSingle.lrSWPosLimitSwitch ) THEN
					xBlockFBFunction:=FALSE;
				END_IF
				IF T_Axis.T_CtrleSingle.lrDistance > 0 AND T_Axis.T_CtrleSingle.xHWLimitNeg THEN
					xBlockFBFunction:=FALSE;
				END_IF
				IF  T_Axis.T_CtrleSingle.lrDistance < 0 AND T_Axis.T_CtrleSingle.xHWLimitPos THEN
					xBlockFBFunction:=FALSE;
				END_IF;
			END_IF;
			IF xMoveVel OR (NOT(T_Axis.T_CtrleSingle.xNotMoving) AND NOT(xMoveAbs) AND NOT(xMoveRel))THEN
				IF ( (T_Axis.T_LiveValue.lrActualPosition >= T_Axis.T_CtrleSingle.lrSWNegLimitSwitch) AND (T_Axis.T_CtrleSingle.lrVelocity < 0) ) OR
				    ( (T_Axis.T_LiveValue.lrActualPosition <= T_Axis.T_CtrleSingle.lrSWPosLimitSwitch) AND (T_Axis.T_CtrleSingle.lrVelocity > 0) ) THEN
					xBlockFBFunction:=FALSE;
				END_IF;
			      IF T_Axis.T_CtrleSingle.lrVelocity > 0 AND T_Axis.T_CtrleSingle.xHWLimitNeg THEN
					xBlockFBFunction:=FALSE;
				END_IF
				IF  T_Axis.T_CtrleSingle.lrVelocity < 0 AND T_Axis.T_CtrleSingle.xHWLimitPos THEN
					xBlockFBFunction:=FALSE;
				END_IF;
			END_IF;
			IF xBlockFBFunction THEN
				xResetAxis:=xReadFile:=xPowerOn:=xPowerOff:=xStop:=	xMoveVel:=xMoveAbs:=xMoveRel:=xHoming:=	xSetPosition:=xCalcAngleRefIndex:=FALSE;
				xSendAxisParameter:=xReadFilePDOMappingPara:=xSendPDOMappingPara:=xMasterSlave:=xSaveParaEcoDrive:=xGetSoftwareVersion:=FALSE;
				xSetSWLimitSwitch:=xResetSWLimitSwitch:=FALSE;
				iStepBlockFunction:=1;
			END_IF;
		END_IF;
		IF xBlockFBFunction THEN
			CASE iStepBlockFunction OF
			1:	IF NOT(SetObjectSDO) THEN
					udiIdxGroup:=16#60FF;	(* Target velocity *)
					udiIndexOffset:=16#0;
					udiLength:=16#4;
					lrReal:=0;
					SetObjectSDO:=TRUE;
					iStepBlockFunction:=iStepBlockFunction+1;
				END_IF;
			2:	IF NOT(SetObjectSDO) THEN
					udiIdxGroup:=16#6081;	(* Profile velocity *)
					udiIndexOffset:=16#0;
					udiLength:=16#4;
					lrReal:=0;
					SetObjectSDO:=TRUE;
					iStepBlockFunction:=iStepBlockFunction+1;
				END_IF;
			3:	IF NOT(SetObjectSDO) THEN
					udiIdxGroup:=16#6060;	(* mode of operation *)
					udiIndexOffset:=16#0;
					udiLength:=16#1;
					lrReal:=1;
					SetObjectSDO:=TRUE;
					iStepBlockFunction:=iStepBlockFunction+1;
				END_IF;
			4:	IF NOT(SetObjectSDO) THEN
					udiIdxGroup:=16#6040;	(* controlword *)
					udiIndexOffset:=16#0;
					udiLength:=16#2;
					lrReal:=16#F;
					SetObjectSDO:=TRUE;
					iStepBlockFunction:=iStepBlockFunction+1;
				END_IF;
			5:	IF NOT(SetObjectSDO) THEN
					xFBErrorActive:=TRUE;
					udiFBErrorID:=16#F213;	(* Limit End Switch Active *)
					xBlockFBFunction:=FALSE;
				END_IF;
			END_CASE;
		END_IF;
	END_IF;

(* Timer *)
	TimerFileLocked(IN:=TRUE, PT:=T#10S);
	TimerFunctionTimeOut(IN:=TRUE,PT:=tTimeOutFunction);

(* detection start *)
	RisingEdgeExecute(CLK:=T_Axis.T_CtrleSingle.xExecute);
	IF RisingEdgeExecute.Q THEN
		CASE T_Axis.T_CtrleSingle.iFunction OF
		(* Reset *)
		1:	xResetAxis:=TRUE;
			iStepResetAxis:=1;
			TimerFunctionTimeOut(IN:=FALSE);
			tTimeOutFunction:=T#7s; (*Verantwortlich für Alarm - Wechsel von iFunction von 1 auf 2 findet nicht statt*)
			xResetController:=FALSE;
		(* Init *)
		2:	xReadFile:=TRUE;
			iStepReadFile:=1;
			TimerFunctionTimeOut(IN:=FALSE);
			tTimeOutFunction:=T#5s;
		(* Power ON *)
		3:	xPowerOn:=TRUE;
			iStepPowerOn:=1;
			TimerFunctionTimeOut(IN:=FALSE);
			tTimeOutFunction:=T#6s;
		(* PowerOff *)
		4:	xPowerOff:=TRUE;
			iStepPowerOff:=1;
			TimerFunctionTimeOut(IN:=FALSE);
			tTimeOutFunction:=T#3s;
		(* Stop *)
		5:	xStop:=TRUE;
			iStepStop:=1;
			TimerFunctionTimeOut(IN:=FALSE);
			tTimeOutFunction:=T#5s;
			xCalcAngleRefIndex:=FALSE;
		(* Move velocity *)
		6:	xMoveVel:=TRUE;
			iStepMoveVel:=1;
			TimerFunctionTimeOut(IN:=FALSE);
			tTimeOutFunction:=T#999999s;
		(* Absolute *)
		7:	xMoveAbs:=TRUE;
			iStepMovePos:=1;
			TimerFunctionTimeOut(IN:=FALSE);
			tTimeOutFunction:=T#999999s;
		(* Relative *)
		8:	xMoveRel:=TRUE;
			iStepMovePos:=1;
			TimerFunctionTimeOut(IN:=FALSE);
			tTimeOutFunction:=T#999999s;
		(* homing *)
		9:	xHoming:=TRUE;
			iStepHoming:=1;
			TimerFunctionTimeOut(IN:=FALSE);
			tTimeOutFunction:=T#999999s;
		(* set position *)
		11:	xSetPosition:=TRUE;
			iStepSetPosition:=1;
			TimerFunctionTimeOut(IN:=FALSE);
			tTimeOutFunction:=T#3s;
		(* calcultate angle between Reference Index and Reference Sensor *)
		19:	xCalcAngleRefIndex:=TRUE;
			iStepCalcAngleRefIndex:=1;
			TimerFunctionTimeOut(IN:=FALSE);
			tTimeOutFunction:=T#999999s;
		(* Send Axis Parameter *)
		21:	xSendAxisParameter:=TRUE;
			iStepSendPara:=1;
			iPtrAxisParameter:=1;
			TimerFunctionTimeOut(IN:=FALSE);
			tTimeOutFunction:=T#5s;
		(* Read Pdo Mapping Parameter *)
		22:	xReadFilePDOMappingPara:=TRUE;
			iStepFile:=1;
			TimerFunctionTimeOut(IN:=FALSE);
			tTimeOutFunction:=T#5s;
		(* Send PDO Mapping Parameter *)
		23: 	xSendPDOMappingPara:=TRUE;
			iStepSendPara:=1;
			iPtrAxisParameter:=1;
			TimerFunctionTimeOut(IN:=FALSE);
			tTimeOutFunction:=T#5s;
		(* Switch Master/Slave *)
		25:	xMasterSlave:=TRUE;
			iStepMasterSlave:=1;
			TimerFunctionTimeOut(IN:=FALSE);
			tTimeOutFunction:=T#3s;
		(* Save Parameter of Servo Drive *)
		26:	xSaveParaEcoDrive:=TRUE;
			iStepSaveParaEcoDrive:=1;
			TimerFunctionTimeOut(IN:=FALSE);
			tTimeOutFunction:=T#3s;
		(* Get Software Version EcoStep *)
		27:	xGetSoftwareVersion:=TRUE;
			iStepGetSoftwareVersion:=1;
			TimerFunctionTimeOut(IN:=FALSE);
			tTimeOutFunction:=T#3s;
		(* Set Software limit switch *)
		28:	xSetSWLimitSwitch:=TRUE;
			iStepSetSWLimitSwitch:=1;
			TimerFunctionTimeOut(IN:=FALSE);
			tTimeOutFunction:=T#3s;
		(* Reset Software limit switch *)
		29:	xResetSWLimitSwitch:=TRUE;
			iStepResetSWLimitSwitch:=1;
			TimerFunctionTimeOut(IN:=FALSE);
			tTimeOutFunction:=T#3s;
		ELSE
		(* function not implemented *)
			xFBErrorActive:=TRUE;
			udiFBErrorID:=16#F201;	(* Function not implemented *)
			(* Exit FB *)
			RETURN;
		END_CASE
		(* Init. variable *)
		T_Axis.T_CtrleSingle.xDone:=FALSE;
		T_Axis.T_CtrleSingle.xErr:=FALSE;
		T_Axis.T_CtrleSingle.udiErrorID:=16#0;
		xConfirmDone:=FALSE;
		xConfirmErr:= FALSE;
		udiConfirmErrorID:=16#0;
		(* Exit FB *)
		RETURN;
	END_IF

(* Reset function *)
	IF xResetAxis THEN
		CASE iStepResetAxis OF
		1:	xResetController:=TRUE;
			xSetEnableAxis:=TRUE;
			iStepResetAxis:=iStepResetAxis+1;
		2:	IF NOT((UINT_TO_WORD(uiStatusWord) AND 16#8) = 16#8) THEN
				xResetController:=FALSE;
				udiIdxGroup:=16#6040;	(* controlword *)
				udiIndexOffset:=16#0;
				udiLength:=16#2;
				lrReal:=16#6;
				SetObjectSDO:=TRUE;
				iStepResetAxis:=iStepResetAxis+1;
			END_IF;
		3:	IF NOT(SetObjectSDO) AND ((UINT_TO_WORD(uiStatusWord) AND 16#31) = 16#31) THEN
				IF NOT(SetObjectSDO) THEN
					udiIdxGroup:=16#60FF;	(* Target velocity *)
					udiIndexOffset:=16#0;
					udiLength:=16#4;
					lrReal:=0;
					SetObjectSDO:=TRUE;
					iStepResetAxis:=iStepResetAxis+1;
				END_IF;
			END_IF;
		4:	IF NOT(SetObjectSDO) THEN
				udiIdxGroup:=16#6081;	(* Profile velocity *)
				udiIndexOffset:=16#0;
				udiLength:=16#4;
				lrReal:=0;
				SetObjectSDO:=TRUE;
				iStepResetAxis:=iStepResetAxis+1;
			END_IF;
		5:	IF NOT(SetObjectSDO) THEN
				udiIdxGroup:=16#6060;	(* mode of operation *)
				udiIndexOffset:=16#0;
				udiLength:=16#1;
				lrReal:=1;
				SetObjectSDO:=TRUE;
				iStepResetAxis:=iStepResetAxis+1;
			END_IF;
		6:	IF NOT(SetObjectSDO) THEN
				udiIdxGroup:=16#2509;	(* Mapping of the speed *)
				udiIndexOffset:=16#2;
				udiLength:=16#4;
				lrReal:=16#0;
				SetObjectSDO:=TRUE;
				iStepResetAxis:=iStepResetAxis+1;
			END_IF;
		7:	IF NOT(SetObjectSDO) THEN
				IF (siOpMode <> 1) THEN
					IF xSetEnableAxis AND xCircuitPowerOn THEN
						udiIdxGroup:=16#6040;	(* controlword *)
						udiIndexOffset:=16#0;
						udiLength:=16#2;
						lrReal:=16#F;
						SetObjectSDO:=TRUE;
						iStepResetAxis:=iStepResetAxis+1;
					ELSE
						iStepResetAxis:=10;
					END_IF;
				ELSE
					iStepResetAxis:=10;
				END_IF;
			END_IF;
		8:	IF NOT(SetObjectSDO) AND ((UINT_TO_WORD(uiStatusWord) AND 16#4037) = 16#4037) THEN
				IF xSetEnableAxis AND xCircuitPowerOn THEN
					udiIdxGroup:=16#6040;	(* controlword *)
					udiIndexOffset:=16#0;
					udiLength:=16#2;
					lrReal:=16#6;
					SetObjectSDO:=TRUE;
					iStepResetAxis:=iStepResetAxis+1;
				ELSE
					iStepResetAxis:=10;
				END_IF;
			END_IF;
		9:	IF NOT(SetObjectSDO) AND ((UINT_TO_WORD(uiStatusWord) AND 16#31) = 16#31) THEN
				iStepResetAxis:=iStepResetAxis+1;
			END_IF;
		10:	IF NOT(SetObjectSDO) THEN
				xSetEnableAxis:=TRUE;
				xNotMoving:=TRUE;
				T_Axis.T_CtrleSingle.xDone:=TRUE;
				T_Axis.T_CtrleSingle.xErr:= FALSE;
				T_Axis.T_CtrleSingle.udiErrorID:=0;
				(* init. variable *)
				xResetAxis:=FALSE;
			END_IF;
		END_CASE;
	END_IF;

(* Init. *)
	IF xReadFile AND NOT(xBlockFBFunction) THEN
		CASE iStepReadFile OF
				(* start timeout *)
		1:	udiFBErrorID:=0;
			(* Check first the usage of the correct parameter *)
			IF (T_Axis.T_Config_Gen.sDeviceFileName = '') THEN
				iStepReadFile:=94;
				RETURN;
			END_IF;
			TimerFileLocked(IN:=FALSE);
			T_Axis.T_FileObj.sData:=sDeleteDataAxis;
			(* next step *)
			iStepReadFile:=iStepReadFile+1;
		(* start read *)
		2:	IF T_HDD.T_Ctrle.xDone AND NOT(T_HDD.T_Ctrle.xLocked) THEN
			(* activ read axis nc parameter *)
				T_HDD.T_Ctrle.xExecute:=TRUE;
				T_HDD.T_Ctrle.xLocked :=TRUE;
				T_HDD.T_Ctrle.iFunction:=1;
				sTmp1:='';
				IF (T_Axis.T_Config_Gen.iMachineType = 1) THEN
					sTmp1:='MicroWire\';
				END_IF;
				IF (T_Axis.T_Config_Gen.iMachineType = 2) THEN
					sTmp1:='MicroRod\';
				END_IF;
				sTmp:='\Hard Disk\Machine450\AxisFile\AxisParameter\';
				sTmp:=CONCAT(sTmp,sTmp1);
				sTmp:=CONCAT(sTmp,T_Axis.T_Config_Gen.sDeviceFileName);
				T_HDD.T_File.sPathAndFileName:=CONCAT(sTmp,'.txt');
				T_HDD.T_Data.sData:=sDeleteDataHDD;
				(* next step *)
				iStepReadFile:=iStepReadFile+1;
			ELSE
			(* activ error if time out done, HDD not ready *)
				IF TimerFileLocked.Q THEN
					 iStepReadFile:=91;
				END_IF
			END_IF
		(* wait done or error *)
		3:	IF T_HDD.T_Ctrle.xDone OR T_HDD.T_Ctrle.xErr THEN
				IF T_HDD.T_Ctrle.xErr  THEN
				(* active step error *)
					iStepReadFile:=92;
				ELSE
				(* next step, init convert value *)
					iStepReadFile:=iStepReadFile+1;
					(* copy data from file *)
					i:=1;
					WHILE T_HDD.T_Data.sData[i] <> '' DO
						T_Axis.T_FileObj.sData[i]:=T_HDD.T_Data.sData[i];
						i:=i+1;
					END_WHILE
					(* erase last line +1 *)
					T_Axis.T_FileObj.sData[i+1]:='';
				END_IF
			END_IF
		(* init. convert *)
		4:	FBConvertAxisParameter(	xStart:=FALSE,
									T_Axis:=T_Axis);
			(* next step, convert value *)
			iStepReadFile:=iStepReadFile+1;
		(* convert value *)
		5:	FBConvertAxisParameter(	xStart:=TRUE,
									T_Axis:=T_Axis);
			IF FBConvertAxisParameter.xDone OR FBConvertAxisParameter.xError THEN
				IF FBConvertAxisParameter.xError THEN
					FBConvertAxisParameter(	xStart:=FALSE,
											T_Axis:=T_Axis);
					(* active step error *)
					iStepReadFile:=93;
				ELSE
					(* activ state read successfull *)
					iStepReadFile:=99;
				END_IF;
			END_IF;
		(* start read error *)
		91:	udiFBErrorID:=16#F202;	(* No HDD free resource, time out *)
			iStepReadFile:=99;
		(* block function error *)
		92:	udiFBErrorID:=16#F203;	(* HDD error, no file found *)
			(* last step *)
			iStepReadFile:=99;
		(* Config File Error *)
		93:	udiFBErrorID:=16#F204;	(* Axis Parameter File, wrong syntax *)
			(* last step *)
			iStepReadFile:=99;
		(* Wrong paramter for this function *)
		94:	udiFBErrorID:=16#F208;	(* Wrong Parameter for Function: Read Axis Parameter *)
			(* last step *)
			iStepReadFile:=99;
		(* init. done *)
		99:	IF T_HDD.T_Ctrle.xErr AND NOT(T_HDD.T_Ctrle.xReset)THEN
				T_HDD.T_Ctrle.xReset:=TRUE;
			END_IF;
			IF (udiFBErrorID <> 0) THEN
				xFBErrorActive:=TRUE;
			END_IF;
			IF NOT(xFBErrorActive) THEN
				T_Axis.T_CtrleSingle.xDone:=TRUE;
				T_Axis.T_CtrleSingle.xErr:= FALSE;
				T_Axis.T_CtrleSingle.udiErrorID:=16#0;
			END_IF;
			xReadFile:=FALSE;
			T_HDD.T_Ctrle.xExecute:=FALSE;
			T_HDD.T_Ctrle.xLocked:=FALSE;
		END_CASE;
	END_IF;

(* Initialisation function *)
	IF xReadFilePDOMappingPara AND NOT(xBlockFBFunction) THEN
		CASE iStepFile OF
		(* start timeout *)
		1:	udiFBErrorID:=0;
			(* Check first the usage of the correct parameter *)
			IF (T_Axis.T_Config_Gen.sFileNamePDOMapping = '') THEN
				iStepFile:=94;
				RETURN;
			END_IF;
			TimerFileLocked(IN:=FALSE);
			T_Axis.T_FileObj.sData:=sDeleteDataAxis;
			(* next step *)
			iStepFile:=iStepFile+1;
		(* start read *)
		2:	IF T_HDD.T_Ctrle.xDone AND NOT(T_HDD.T_Ctrle.xLocked) THEN
			(* activ read axis nc parameter *)
				T_HDD.T_Ctrle.xExecute:=TRUE;
				T_HDD.T_Ctrle.xLocked :=TRUE;
				T_HDD.T_Ctrle.iFunction:=1;
				sTmp:='\Hard Disk\Machine450\AxisFile\PDOMapping\';
				sTmp:=CONCAT(sTmp,T_Axis.T_Config_Gen.sFileNamePDOMapping);
				T_HDD.T_File.sPathAndFileName:=CONCAT(sTmp,'.txt');
				T_HDD.T_Data.sData:=sDeleteDataHDD;
				(* next step *)
				iStepFile:=iStepFile+1;
			ELSE
			(* activ error if time out done, HDD not ready *)
				IF TimerFileLocked.Q THEN
					 iStepFile:=91;
				END_IF
			END_IF
		(* wait done or error *)
		3:	IF T_HDD.T_Ctrle.xDone OR T_HDD.T_Ctrle.xErr THEN
				IF T_HDD.T_Ctrle.xErr  THEN
				(* active step error *)
					iStepFile:=92;
				ELSE
				(* next step, init convert value *)
					iStepFile:=iStepFile+1;
					(* copy data from file *)
					i:=1;
					WHILE T_HDD.T_Data.sData[i] <> '' DO
						T_Axis.T_FileObj.sData[i]:=T_HDD.T_Data.sData[i];
						i:=i+1;
					END_WHILE
					(* erase last line +1 *)
					T_Axis.T_FileObj.sData[i+1]:='';
				END_IF
			END_IF
		(* init. convert *)
		4:	FBConvertPdoMapping(	xStart:=FALSE,
								T_Axis:=T_Axis);
			(* next step, convert value *)
			iStepFile:=iStepFile+1;
		(* convert value *)
		5:	FBConvertPdoMapping(	xStart:=TRUE,
									T_Axis:=T_Axis);
			IF FBConvertPdoMapping.xDone OR FBConvertPdoMapping.xError THEN
				IF FBConvertPdoMapping.xError THEN
					FBConvertPdoMapping(	xStart:=FALSE,
											T_Axis:=T_Axis);
					(* active step error *)
					iStepFile:=93;
				ELSE
					(* activ state read successfull *)
					iStepFile:=99;
				END_IF;
			END_IF;
		(* start read error *)
		91:	udiFBErrorID:=16#F202;	(* No HDD free resource, time out *)
			iStepFile:=99;
		(* block function error *)
		92:	udiFBErrorID:=16#F203;	(* HDD error, no file found *)
			(* last step *)
			iStepFile:=99;
		(* Config File Error *)
		93:	udiFBErrorID:=16#F205;	(* PDOMapping Parameter File, wrong syntax *)
			(* last step *)
			iStepFile:=99;
		(* Wrong paramter for this function *)
		94:	udiFBErrorID:=16#F209;	(* Wrong Parameter for Function: Read PDOMapping Parameter *)
			(* last step *)
			iStepFile:=99;
		(* init. done *)
		99:	IF T_HDD.T_Ctrle.xErr AND NOT(T_HDD.T_Ctrle.xReset)THEN
				T_HDD.T_Ctrle.xReset:=TRUE;
			END_IF;
			IF (udiFBErrorID <> 0) THEN
				xFBErrorActive:=TRUE;
			END_IF;
			IF NOT(xFBErrorActive) THEN
				T_Axis.T_CtrleSingle.xDone:=TRUE;
				T_Axis.T_CtrleSingle.xErr:= FALSE;
				T_Axis.T_CtrleSingle.udiErrorID:=16#0;
			END_IF;
			xReadFilePDOMappingPara:=FALSE;
			T_HDD.T_Ctrle.xExecute:=FALSE;
			T_HDD.T_Ctrle.xLocked:=FALSE;
		END_CASE
	END_IF

(* Power function On/Off *)
	RisingEdgePowerOn(CLK:=xPowerOn);
	RisingEdgePowerOff(CLK:=xPowerOff);
	IF xPowerOn AND NOT(xBlockFBFunction) THEN
		CASE iStepPowerOn OF
		1:	IF xSetEnableAxis AND xCircuitPowerOn THEN
				udiIdxGroup:=16#6040;	(* controlword *)
				udiIndexOffset:=16#0;
				udiLength:=16#2;
				lrReal:=16#F;
				SetObjectSDO:=TRUE;
				iStepPowerOn:=iStepPowerOn+1;
			ELSE
				xFBErrorActive:=TRUE;
				udiFBErrorID:=16#F207;	(* No Axis Power Supply *)
			END_IF;
		2:	IF NOT(SetObjectSDO) AND ((UINT_TO_WORD(uiStatusWord) AND 16#4037) = 16#4037) THEN
				T_Axis.T_CtrleSingle.xDone:=TRUE;
				T_Axis.T_CtrleSingle.xErr:= FALSE;
				T_Axis.T_CtrleSingle.udiErrorID:=0;
				(* init. variable *)
				xPowerOn:=FALSE;
				xNotMoving:=TRUE;
			END_IF;
		END_CASE;
	END_IF
	IF xPowerOff AND NOT(xBlockFBFunction) THEN
		CASE iStepPowerOff OF
		1:	IF xSetEnableAxis AND xCircuitPowerOn THEN
				udiIdxGroup:=16#6040;	(* controlword *)
				udiIndexOffset:=16#0;
				udiLength:=16#2;
				lrReal:=16#6;
				SetObjectSDO:=TRUE;
				iStepPowerOff:=iStepPowerOff+1;
			ELSE
				xFBErrorActive:=TRUE;
				udiFBErrorID:=16#F207;	(* No Axis Power Supply *)
			END_IF;
		2:	IF NOT(SetObjectSDO) AND ((UINT_TO_WORD(uiStatusWord) AND 16#31) = 16#31) THEN
				T_Axis.T_CtrleSingle.xDone:=TRUE;
				T_Axis.T_CtrleSingle.xErr:= FALSE;
				T_Axis.T_CtrleSingle.udiErrorID:=0;
				(* init. variable *)
				xPowerOff:=FALSE;
				xNotMoving:=TRUE;
			END_IF;
		END_CASE;
	END_IF

(* Stop function *)
	RisingEdgeStop(CLK:=xStop);
	IF xStop AND NOT(xBlockFBFunction) THEN
		CASE iStepStop OF
		1:	IF xNotMoving AND NOT(xMoveAbs) AND NOT(xMoveRel) AND NOT(xMoveVel) AND NOT(xHoming) THEN
				iStepStop:=9;
				xMoveAbs:=xMoveRel:=xMoveVel:=xHoming:=FALSE;
				RETURN;
			END_IF;
			IF (siOpMode = 3) THEN
				IF NOT(SetObjectSDO) AND NOT(GetObjectSDO) THEN
					udiIdxGroup:=16#60FF;	(* Target velocity *)
					udiIndexOffset:=16#0;
					udiLength:=16#4;
					lrReal:=0;
					SetObjectSDO:=TRUE;
					iStepStop:=2;
					xMoveAbs:=xMoveRel:=xMoveVel:=xHoming:=FALSE;
				END_IF;
			END_IF;
			IF (siOpMode = 1) AND (xMoveAbs OR xMoveRel) THEN
				IF NOT(SetObjectSDO) AND NOT(GetObjectSDO) THEN
					udiIdxGroup:=16#6081;	(* Profile velocity *)
					udiIndexOffset:=16#0;
					udiLength:=16#4;
					lrReal:=0;
					SetObjectSDO:=TRUE;
					iStepStop:=3;
					xMoveAbs:=xMoveRel:=xMoveVel:=xHoming:=FALSE;
				END_IF;
			END_IF;
			IF (siOpMode = 6) AND xHoming THEN
				IF NOT(SetObjectSDO) AND NOT(GetObjectSDO) THEN
					udiIdxGroup:=16#6040;	(* controlword *)
					udiIndexOffset:=16#0;
					udiLength:=16#2;
					lrReal:=16#F;
					SetObjectSDO:=TRUE;
					iStepStop:=7;
					WaitSwitchReady(IN:=FALSE);
					xMoveAbs:=xMoveRel:=xMoveVel:=xHoming:=FALSE;
				END_IF;
			END_IF;
(*
			IF (xMoveAbs OR xMoveRel) AND (iStepStop = 1) THEN
				iStepStop:=9;
				RETURN;
			END_IF;
*)
		2:	IF NOT(SetObjectSDO) AND GETBIT32(uiStatusWord,12) THEN
				udiIdxGroup:=16#6060;	(* mode of operation *)
				udiIndexOffset:=16#0;
				udiLength:=16#1;
				lrReal:=1;
				SetObjectSDO:=TRUE;
				iStepStop:=10;
			END_IF;
		3:	IF NOT(SetObjectSDO) THEN
				udiIdxGroup:=16#60FF;	(* Target velocity *)
				udiIndexOffset:=16#0;
				udiLength:=16#4;
				lrReal:=0;
				SetObjectSDO:=TRUE;
				iStepStop:=4;
			END_IF;
		4:	IF NOT(SetObjectSDO) THEN
				udiIdxGroup:=16#6060;	(* mode of operation *)
				udiIndexOffset:=16#0;
				udiLength:=16#1;
				lrReal:=3;
				SetObjectSDO:=TRUE;
				iStepStop:=5;
			END_IF;
		5:	IF NOT(SetObjectSDO) AND ((UINT_TO_WORD(uiStatusWord) AND 16#1400) = 16#1400) THEN
				udiIdxGroup:=16#6040;	(* controlword *)
				udiIndexOffset:=16#0;
				udiLength:=16#2;
				lrReal:=16#F;
				SetObjectSDO:=TRUE;
				iStepStop:=6;
			END_IF;
		6:	IF NOT(SetObjectSDO) THEN
				udiIdxGroup:=16#6060;	(* mode of operation *)
				udiIndexOffset:=16#0;
				udiLength:=16#1;
				lrReal:=1;
				SetObjectSDO:=TRUE;
				iStepStop:=9;
			END_IF;
		7:	WaitSwitchReady(IN:=TRUE,PT:=T#1000ms);
			IF WaitSwitchReady.Q THEN
				IF NOT(SetObjectSDO) THEN
					WaitSwitchReady(IN:=FALSE);
					udiIdxGroup:=16#6060;	(* mode of operation *)
					udiIndexOffset:=16#0;
					udiLength:=16#1;
					lrReal:=3;
					SetObjectSDO:=TRUE;
					iStepStop:=8;
				END_IF;
			END_IF;
		8:	IF NOT(SetObjectSDO) AND ((UINT_TO_WORD(uiStatusWord) AND 16#1400) = 16#1400) THEN
				udiIdxGroup:=16#6060;	(* mode of operation *)
				udiIndexOffset:=16#0;
				udiLength:=16#1;
				lrReal:=1;
				SetObjectSDO:=TRUE;
				iStepStop:=9;
			END_IF;
		9:	IF NOT(SetObjectSDO) THEN
				IF NOT(xCalcAngleRefIndex) THEN
					T_Axis.T_CtrleSingle.xDone:=TRUE;
					T_Axis.T_CtrleSingle.xErr:= FALSE;
					T_Axis.T_CtrleSingle.udiErrorID:=0;
				END_IF;
				(* init. variable *)
				xStop:=FALSE;
				xNotMoving:=TRUE;
			END_IF;
		10:	IF NOT(SetObjectSDO) AND ((UINT_TO_WORD(uiStatusWord) AND 16#1000) = 16#1000) THEN
				IF NOT(xCalcAngleRefIndex) THEN
					T_Axis.T_CtrleSingle.xDone:=TRUE;
					T_Axis.T_CtrleSingle.xErr:= FALSE;
					T_Axis.T_CtrleSingle.udiErrorID:=0;
				END_IF;
				(* init. variable *)
				xStop:=FALSE;
				xNotMoving:=TRUE;
			END_IF;
		END_CASE;
	END_IF;

(* Move velocity *)
	IF xMoveVel AND NOT(xBlockFBFunction) THEN
		CASE iStepMoveVel OF
		1:	udiFBErrorID:=0;
			(* Check first the usage of the correct parameter *)
			IF (T_Axis.T_CtrleSingle.lrAcceleration = 0) OR (T_Axis.T_CtrleSingle.lrDecceleration = 0) OR (T_Axis.T_CtrleSingle.lrVelocity = 0) THEN
				iStepMoveVel:=91;
				RETURN;
			END_IF;
			(* Check if the power supply of the Axis is on *)
			IF NOT(T_Axis.T_CtrleSingle.xPower) THEN
				iStepMoveVel:=92;
				RETURN;
			END_IF;
			udiIdxGroup:=16#6083;	(* Acceleration *)
			udiIndexOffset:=16#0;
			udiLength:=16#4;
			lrReal:=T_Axis.T_CtrleSingle.lrAcceleration * T_Axis.T_CtrleSingle.lrScaleFactor * 64.0;
			SetObjectSDO:=TRUE;
			iStepMoveVel:=iStepMoveVel+1;
			xNotMoving:=TRUE;
		2:	IF NOT(SetObjectSDO) THEN
				udiIdxGroup:=16#6084;	(* Deceleration *)
				udiIndexOffset:=16#0;
				udiLength:=16#4;
				lrReal:=T_Axis.T_CtrleSingle.lrDecceleration * T_Axis.T_CtrleSingle.lrScaleFactor * 64.0;
				SetObjectSDO:=TRUE;
				iStepMoveVel:=iStepMoveVel+1;
			END_IF;
		3:	IF NOT(SetObjectSDO) THEN
				IF (siOpMode <> 3) THEN
					udiIdxGroup:=16#6060;	(* mode of operation *)
					udiIndexOffset:=16#0;
					udiLength:=16#1;
					lrReal:=3;
					SetObjectSDO:=TRUE;
				END_IF;
				iStepMoveVel:=iStepMoveVel+1;
			END_IF;
		4:	IF NOT(SetObjectSDO) THEN
				udiIdxGroup:=16#60FF;	(* Target velocity *)
				udiIndexOffset:=16#0;
				udiLength:=16#4;
				IF (T_Axis.T_Config_Gen.iTyp = 1) OR (T_Axis.T_Config_Gen.iTyp = 2) OR (T_Axis.T_Config_Gen.iTyp = 3) THEN
					lrReal:=((T_Axis.T_CtrleSingle.lrVelocity/60.0) * 64.0) * (360.0 * T_Axis.T_CtrleSingle.lrScaleFactor);
				ELSE
					lrReal:=T_Axis.T_CtrleSingle.lrVelocity * T_Axis.T_CtrleSingle.lrScaleFactor * 64.0;
				END_IF;
				SetObjectSDO:=TRUE;
				iStepMoveVel:=iStepMoveVel+1;
			END_IF;
		5:	IF NOT(SetObjectSDO) AND NOT(GETBIT32(uiStatusWord,12)) THEN
				iStepMoveVel:=99;
			END_IF;
		(* Wrong paramter for this function *)
		91:	udiFBErrorID:=16#F20A;	(* Wrong Parameter for Function: Move velocity *)
			(* last step *)
			iStepMoveVel:=99;
		(* No power supply of the Axis *)
		92:	udiFBErrorID:=16#F212;	(* Can't move, no power supply *)
			(* last step *)
			iStepMoveVel:=99;
		(* init. done *)
		99:	IF (udiFBErrorID <> 0) THEN
				xFBErrorActive:=TRUE;
			END_IF;
			IF NOT(xFBErrorActive) THEN
				T_Axis.T_CtrleSingle.xDone:=TRUE;
				T_Axis.T_CtrleSingle.xErr:= FALSE;
				T_Axis.T_CtrleSingle.udiErrorID:=16#0;
			END_IF;
			(* init. variable *)
			xMoveVel:=FALSE;
			xNotMoving:=FALSE;
		END_CASE;
	END_IF

(* Move to position ABS/Rel *)
	IF (xMoveAbs OR xMoveRel) AND NOT(xBlockFBFunction) THEN
		CASE iStepMovePos OF
		1:	udiFBErrorID:=0;
			(* Check first the usage of the correct parameter *)
			IF (T_Axis.T_CtrleSingle.lrAcceleration = 0) OR (T_Axis.T_CtrleSingle.lrDecceleration = 0) OR (T_Axis.T_CtrleSingle.lrVelocity = 0) (*OR
			     ((T_Axis.T_CtrleSingle.lrDistance = 0) AND xMoveRel) *)THEN
				iStepMovePos:=91;
				RETURN;
			END_IF;
			(* Check if the power supply of the Axis is on *)
			IF NOT(T_Axis.T_CtrleSingle.xPower) THEN
				iStepMovePos:=92;
				RETURN;
			END_IF;
			udiIdxGroup:=16#6040;	(* Controlword *)
			udiIndexOffset:=16#0;
			udiLength:=16#2;
			lrReal:=16#F;
			SetObjectSDO:=TRUE;
			IF T_Axis.T_CtrleSingle.xBlockAcclDeclParameter THEN
				T_Axis.T_CtrleSingle.xBlockAcclDeclParameter:=FALSE;
				IF (siOpMode = 1) THEN
					iStepMovePos:=iStepMovePos+4;
				ELSE
					iStepMovePos:=iStepMovePos+3;
				END_IF;
			ELSE
				iStepMovePos:=iStepMovePos+1;
			END_IF;
			xNotMoving:=TRUE;
		2:	IF NOT(SetObjectSDO) THEN
				udiIdxGroup:=16#6083;	(* Acceleration *)
				udiIndexOffset:=16#0;
				udiLength:=16#4;
				lrReal:=T_Axis.T_CtrleSingle.lrAcceleration * T_Axis.T_CtrleSingle.lrScaleFactor * 64.0;
				SetObjectSDO:=TRUE;
				iStepMovePos:=iStepMovePos+1;
			END_IF;
		3:	IF NOT(SetObjectSDO) THEN
				udiIdxGroup:=16#6084;	(* Deceleration *)
				udiIndexOffset:=16#0;
				udiLength:=16#4;
				lrReal:=T_Axis.T_CtrleSingle.lrDecceleration * T_Axis.T_CtrleSingle.lrScaleFactor * 64.0;
				SetObjectSDO:=TRUE;
				iStepMovePos:=iStepMovePos+1;
			END_IF;
		4:	IF NOT(SetObjectSDO) THEN
				IF (siOpMode <> 1) THEN
					udiIdxGroup:=16#6060;	(* mode of operation *)
					udiIndexOffset:=16#0;
					udiLength:=16#1;
					lrReal:=1;
					SetObjectSDO:=TRUE;
				END_IF;
				iStepMovePos:=iStepMovePos+1;
			END_IF;
		5:	IF NOT(SetObjectSDO) THEN
				udiIdxGroup:=16#607A;	(* Target position *)
				udiIndexOffset:=16#0;
				udiLength:=16#4;
				IF xMoveAbs THEN
					IF (T_Axis.T_Config_Gen.iTyp <> 5) THEN
						lrReal:=T_Axis.T_CtrleSingle.lrPosition * T_Axis.T_CtrleSingle.lrScaleFactor;
					ELSE
						lrReal:=T_Axis.T_CtrleSingle.lrPosition * T_Axis.T_CtrleSingle.lrScaleFactor * rPrismaFactor;
					END_IF;
				END_IF;
				IF xMoveRel THEN
					IF (T_Axis.T_Config_Gen.iTyp <> 5) THEN
						lrReal:=T_Axis.T_CtrleSingle.lrDistance * T_Axis.T_CtrleSingle.lrScaleFactor;
					ELSE
						lrReal:=T_Axis.T_CtrleSingle.lrDistance * T_Axis.T_CtrleSingle.lrScaleFactor * rPrismaFactor;
					END_IF;
				END_IF;
				SetObjectSDO:=TRUE;
				iStepMovePos:=iStepMovePos+1;
			END_IF;
		6:	IF NOT(SetObjectSDO) THEN
				udiIdxGroup:=16#6081;	(* Profile velocity *)
				udiIndexOffset:=16#0;
				udiLength:=16#4;
				IF (T_Axis.T_Config_Gen.iTyp = 1) OR (T_Axis.T_Config_Gen.iTyp = 2) OR (T_Axis.T_Config_Gen.iTyp = 3) THEN
					lrReal:=((ABS(T_Axis.T_CtrleSingle.lrVelocity)/60.0) * 64.0) * (360.0 * T_Axis.T_CtrleSingle.lrScaleFactor);
				ELSE
					IF (T_Axis.T_Config_Gen.iTyp = 5) THEN
						lrReal:=ABS(T_Axis.T_CtrleSingle.lrVelocity) * T_Axis.T_CtrleSingle.lrScaleFactor * 64.0 * rPrismaFactor;
					ELSE
						lrReal:=ABS(T_Axis.T_CtrleSingle.lrVelocity) * T_Axis.T_CtrleSingle.lrScaleFactor * 64.0;
					END_IF;
				END_IF;
				lrForceSpeed:=lrReal;
				SetObjectSDO:=TRUE;
				iStepMovePos:=iStepMovePos+1;
			END_IF;
		7:	IF NOT(SetObjectSDO) THEN
				udiIdxGroup:=16#6040;	(* controlword *)
				udiIndexOffset:=16#0;
				udiLength:=16#2;
				IF xMoveAbs THEN
					lrReal:=16#3F;
				END_IF;
				IF xMoveRel THEN
					lrReal:=16#7F;
				END_IF;
				SetObjectSDO:=TRUE;
				iStepMovePos:=iStepMovePos+1;
				xNotMoving:=FALSE;
			END_IF;
		8:	IF NOT(SetObjectSDO) AND ((UINT_TO_WORD(uiStatusWord) AND 16#1400) = 16#1400) THEN
				udiIdxGroup:=16#6040;	(* Controlword *)
				udiIndexOffset:=16#0;
				udiLength:=16#2;
				lrReal:=16#F;
				SetObjectSDO:=TRUE;
				iStepMovePos:=iStepMovePos+1;
				xNotMoving:=FALSE;
			END_IF;
		9:	IF NOT(SetObjectSDO) AND ((UINT_TO_WORD(uiStatusWord) AND 16#4037) = 16#4037) THEN
				iStepMovePos:=99;
			END_IF;
		(* Wrong paramter for this function *)
		91:	IF xMoveAbs THEN
				udiFBErrorID:=16#F20B;	(* Wrong Parameter for Function: Move position absolute *)
			END_IF;
			IF xMoveRel THEN
				udiFBErrorID:=16#F20C;	(* Wrong Parameter for Function: Move position relative *)
			END_IF;
			(* last step *)
			iStepMovePos:=99;
		(* No power supply of the Axis *)
		92:	udiFBErrorID:=16#F212;	(* Can't move, no power supply *)
			(* last step *)
			iStepMovePos:=99;
		(* init. done *)
		99:	IF (udiFBErrorID <> 0)  THEN
				xFBErrorActive:=TRUE;
				xCalcAngleRefIndex:=FALSE;
			END_IF;
			IF NOT(xFBErrorActive) AND NOT(xCalcAngleRefIndex) THEN
				T_Axis.T_CtrleSingle.xDone:=TRUE;
				T_Axis.T_CtrleSingle.xErr:= FALSE;
				T_Axis.T_CtrleSingle.udiErrorID:=16#0;
			END_IF;
			(* init. variable *)
			xMoveAbs:=xMoveRel:=FALSE;
			xNotMoving:=TRUE;
		END_CASE;
	END_IF;

(* Homing *)
	IF xHoming AND NOT(xBlockFBFunction) THEN
		CASE iStepHoming OF
		1:	udiFBErrorID:=0;
			(* Check first the usage of the correct parameter *)
			IF (T_Axis.T_CtrleSingle.lrHomingMethode <= 0) OR (T_Axis.T_CtrleSingle.lrHomingMethode > 34) OR (T_Axis.T_CtrleSingle.lrHomeSpeedSwitch = 0) OR
			     (T_Axis.T_CtrleSingle.lrHomeSpeedZero = 0) OR (T_Axis.T_CtrleSingle.lrHomeAcceleration = 0) THEN
				iStepHoming:=91;
				RETURN;
			END_IF;
			(* Check if the power supply of the Axis is on *)
			IF NOT(T_Axis.T_CtrleSingle.xPower) THEN
				iStepHoming:=92;
				RETURN;
			END_IF;
			udiIdxGroup:=16#6040;	(* Controlword *)
			udiIndexOffset:=16#0;
			udiLength:=16#2;
			lrReal:=16#F;
			SetObjectSDO:=TRUE;
			iStepHoming:=iStepHoming+1;
			xNotMoving:=TRUE;
		2:	IF NOT(SetObjectSDO) THEN
				IF (siOpMode <> 1) THEN
					udiIdxGroup:=16#6060;	(* mode of operation *)
					udiIndexOffset:=16#0;
					udiLength:=16#1;
					lrReal:=1;
					SetObjectSDO:=TRUE;
					iStepHoming:=iStepHoming+1;
					TONWaitSetValue(IN:=FALSE);
				ELSE
					iStepHoming:=iStepHoming+2;
				END_IF;
			END_IF;
		3:	IF NOT(SetObjectSDO) THEN
				TONWaitSetValue(IN:=TRUE,PT:=T#100ms);
				IF TONWaitSetValue.Q THEN
					TONWaitSetValue(IN:=FALSE);
					iStepHoming:=iStepHoming+1;
				END_IF;
			END_IF;
		4:	IF NOT(SetObjectSDO) THEN
				(* It is Important that the accl. for the homing is settled before the mode of operation is set to the homing, otherwise it will not work with this accl. *)
				udiIdxGroup:=16#609A;	(* homing acceleration *)
				udiIndexOffset:=16#0;
				udiLength:=16#4;
				lrReal:=T_Axis.T_CtrleSingle.lrHomeAcceleration * T_Axis.T_CtrleSingle.lrScaleFactor * 64.0;
				SetObjectSDO:=TRUE;
				iStepHoming:=iStepHoming+1;
			END_IF;
		5:	IF NOT(SetObjectSDO) THEN
				udiIdxGroup:=16#6083;	(* Acceleration *)
				udiIndexOffset:=16#0;
				udiLength:=16#4;
				lrReal:=T_Axis.T_CtrleSingle.lrAcceleration * T_Axis.T_CtrleSingle.lrScaleFactor * 64.0;
				SetObjectSDO:=TRUE;
				iStepHoming:=iStepHoming+1;
			END_IF;
		6:	IF NOT(SetObjectSDO) THEN
				udiIdxGroup:=16#6084;	(* Deceleration *)
				udiIndexOffset:=16#0;
				udiLength:=16#4;
				lrReal:=T_Axis.T_CtrleSingle.lrDecceleration * T_Axis.T_CtrleSingle.lrScaleFactor * 64.0;
				SetObjectSDO:=TRUE;
				iStepHoming:=iStepHoming+1;
				TONWaitSetValue(IN:=FALSE);
			END_IF;
		7:	IF NOT(SetObjectSDO) THEN
				TONWaitSetValue(IN:=TRUE,PT:=T#200ms);
				IF TONWaitSetValue.Q THEN
					TONWaitSetValue(IN:=FALSE);
					iStepHoming:=iStepHoming+1;
				END_IF;
			END_IF;
		8:	IF NOT(SetObjectSDO) THEN
				IF (siOpMode <> 6) THEN
					udiIdxGroup:=16#6060;	(* mode of operation *)
					udiIndexOffset:=16#0;
					udiLength:=16#1;
					lrReal:=6;
					SetObjectSDO:=TRUE;
				END_IF;
				iStepHoming:=iStepHoming+1;
			END_IF;
		9:	IF NOT(SetObjectSDO) THEN
				udiIdxGroup:=16#6098;	(* Homing Methode *)
				udiIndexOffset:=16#0;
				udiLength:=16#1;
				lrReal:=T_Axis.T_CtrleSingle.lrHomingMethode;
				SetObjectSDO:=TRUE;
				iStepHoming:=iStepHoming+1;
			END_IF;

		10:	IF NOT(SetObjectSDO) THEN
				udiIdxGroup:=16#607C;	(* Home Offset *)
				udiIndexOffset:=16#0;
				udiLength:=16#4;
				lrReal:=T_Axis.T_CtrleSingle.lrHomeOffset * T_Axis.T_CtrleSingle.lrScaleFactor ;
				SetObjectSDO:=TRUE;
				iStepHoming:=iStepHoming+1;
			END_IF;
		11:	IF NOT(SetObjectSDO) THEN
				udiIdxGroup:=16#6099;	(* homing speed search for switch *)
				udiIndexOffset:=16#1;
				udiLength:=16#4;
				lrReal:=T_Axis.T_CtrleSingle.lrHomeSpeedSwitch * T_Axis.T_CtrleSingle.lrScaleFactor * 64.0;
				SetObjectSDO:=TRUE;
				iStepHoming:=iStepHoming+1;
			END_IF;
		12:	IF NOT(SetObjectSDO) THEN
				udiIdxGroup:=16#6099;	(* homing speed search for zero *)
				udiIndexOffset:=16#2;
				udiLength:=16#4;
				lrReal:=T_Axis.T_CtrleSingle.lrHomeSpeedZero * T_Axis.T_CtrleSingle.lrScaleFactor * 64.0;
				SetObjectSDO:=TRUE;
				iStepHoming:=iStepHoming+1;
			END_IF;
		13:	IF NOT(SetObjectSDO) THEN
				udiIdxGroup:=16#6040;	(* controlword *)
				udiIndexOffset:=16#0;
				udiLength:=16#2;
				lrReal:=16#1F;
				SetObjectSDO:=TRUE;
				iStepHoming:=iStepHoming+1;
			END_IF;
		14:	IF NOT(SetObjectSDO) AND ((UINT_TO_WORD(uiStatusWord) AND 16#1400) = 16#1400) THEN
				udiIdxGroup:=16#6040;	(* Controlword *)
				udiIndexOffset:=16#0;
				udiLength:=16#2;
				lrReal:=16#F;
				SetObjectSDO:=TRUE;
				iStepHoming:=iStepHoming+1;
				xNotMoving:=FALSE;
			END_IF;
		15:	IF NOT(SetObjectSDO) AND ((UINT_TO_WORD(uiStatusWord) AND 16#4037) = 16#4037) THEN
				iStepHoming:=99;
			END_IF;
		(* Wrong paramter for this function *)
		91:	udiFBErrorID:=16#F20D;	(* Wrong Parameter for Function: Move referencing *)
			(* last step *)
			iStepHoming:=99;
		(* No power supply of the Axis *)
		92:	udiFBErrorID:=16#F212;	(* Can't move, no power supply *)
			(* last step *)
			iStepHoming:=99;
		(* init. done *)
		99:	IF (udiFBErrorID <> 0) THEN
				xFBErrorActive:=TRUE;
				xCalcAngleRefIndex:=FALSE;
			END_IF;
			IF NOT(xFBErrorActive) AND NOT(xCalcAngleRefIndex) THEN
				T_Axis.T_CtrleSingle.xDone:=TRUE;
				T_Axis.T_CtrleSingle.xErr:= FALSE;
				T_Axis.T_CtrleSingle.udiErrorID:=16#0;
			END_IF;
			(* init. variable *)
			xHoming:=FALSE;
			xNotMoving:=TRUE;
		END_CASE;
	END_IF;

(* Set new position *)
	IF xSetPosition AND NOT(xBlockFBFunction) THEN
		CASE iStepSetPosition OF
		1:	udiIdxGroup:=16#6040;	(* Controlword *)
			udiIndexOffset:=16#0;
			udiLength:=16#2;
			lrReal:=16#F;
			SetObjectSDO:=TRUE;
			iStepSetPosition:=iStepSetPosition+1;
		2:	IF NOT(SetObjectSDO) THEN
				IF (siOpMode <> 6) THEN
					udiIdxGroup:=16#6060;	(* mode of operation *)
					udiIndexOffset:=16#0;
					udiLength:=16#1;
					lrReal:=6;
					SetObjectSDO:=TRUE;
				END_IF;
				iStepSetPosition:=iStepSetPosition+1;
			END_IF;
		3:	IF NOT(SetObjectSDO) THEN
				udiIdxGroup:=16#6098;	(* Homing Methode *)
				udiIndexOffset:=16#0;
				udiLength:=16#1;
				lrReal:=34;			(* Referenzmethode 34 without Referenzdrive *)
				SetObjectSDO:=TRUE;
				iStepSetPosition:=iStepSetPosition+1;
			END_IF;
		4:	IF NOT(SetObjectSDO) THEN
				udiIdxGroup:=16#607C;	(* Home Offset *)
				udiIndexOffset:=16#0;
				udiLength:=16#4;
				IF (T_Axis.T_Config_Gen.iTyp <> 5) THEN
					lrReal:=T_Axis.T_CtrleSingle.rSetPosition * T_Axis.T_CtrleSingle.lrScaleFactor * -1.0;
				ELSE
					lrReal:=T_Axis.T_CtrleSingle.rSetPosition * T_Axis.T_CtrleSingle.lrScaleFactor * rPrismaFactor * -1.0;
				END_IF;
				SetObjectSDO:=TRUE;
				iStepSetPosition:=iStepSetPosition+1;
			END_IF;
		5:	IF NOT(SetObjectSDO) THEN
				udiIdxGroup:=16#6040;	(* controlword *)
				udiIndexOffset:=16#0;
				udiLength:=16#2;
				lrReal:=16#1F;
				SetObjectSDO:=TRUE;
				iStepSetPosition:=iStepSetPosition+1;
			END_IF;
		6:	IF NOT(SetObjectSDO) AND ((UINT_TO_WORD(uiStatusWord) AND 16#1400) = 16#1400) THEN
				udiIdxGroup:=16#6040;	(* Controlword *)
				udiIndexOffset:=16#0;
				udiLength:=16#2;
				lrReal:=16#F;
				SetObjectSDO:=TRUE;
				iStepSetPosition:=iStepSetPosition+1;
			END_IF;
		7:	IF NOT(SetObjectSDO) AND ((UINT_TO_WORD(uiStatusWord) AND 16#4037) = 16#4037) THEN
				T_Axis.T_CtrleSingle.xDone:=TRUE;
				T_Axis.T_CtrleSingle.xErr:= FALSE;
				T_Axis.T_CtrleSingle.udiErrorID:=0;
				(* init. variable *)
				xSetPosition:=FALSE;
			END_IF;
		END_CASE;
	END_IF;

(* calcultate angle between Reference Index and Reference Sensor *)
	IF xCalcAngleRefIndex AND NOT(xBlockFBFunction) THEN
		CASE iStepCalcAngleRefIndex OF
		1:	udiFBErrorID:=0;
			xHoming:=TRUE;
			iStepHoming:=1;
			T_Axis.T_CtrleSingle.iStrokeAngleRefIndex:=0;
			iStepCalcAngleRefIndex:=iStepCalcAngleRefIndex + 1;
		2:	IF NOT(xHoming) THEN
				xMoveAbs:=TRUE;
				iStepMovePos:=1;
				iStepCalcAngleRefIndex:=iStepCalcAngleRefIndex + 1;
			END_IF;
		3:	IF NOT(xMoveAbs) THEN
				xMoveRel:=TRUE;
				iStepMovePos:=1;
				iStepCalcAngleRefIndex:=iStepCalcAngleRefIndex + 1;
			END_IF;
		4:	IF NOT(xMoveRel) THEN
				iStepCalcAngleRefIndex:=91;
			END_IF;
			IF GETBIT32(T_Axis.T_TxPdoParameter.udiDigitalInput,23) THEN
				lrCapturePosition:=ABS(T_Axis.T_LiveValue.lrActualPosition);
				xStop:=TRUE;
				iStepStop:=1;
				iStepCalcAngleRefIndex:=iStepCalcAngleRefIndex + 1;
			END_IF;
		5:	IF NOT(xStop) THEN
				T_Axis.T_CtrleSingle.iStrokeAngleRefIndex:=LREAL_TO_INT((360.0/8000.0) * lrCapturePosition * T_Axis.T_CtrleSingle.lrScaleFactor);	(* calculate Distance between RefSensor and RefIndex *)
				iStepCalcAngleRefIndex:=99;
			END_IF;
		(* Wrong paramter for this function *)
		91:	udiFBErrorID:=16#F211;	(* Function CalcAnlgeRefIndex:Ref.Sensor not found *)
			(* last step *)
			iStepCalcAngleRefIndex:=99;
		(* init. done *)
		99:	IF (udiFBErrorID <> 0)  THEN
				xFBErrorActive:=TRUE;
			END_IF;
			IF NOT(xFBErrorActive) THEN
				T_Axis.T_CtrleSingle.xDone:=TRUE;
				T_Axis.T_CtrleSingle.xErr:= FALSE;
				T_Axis.T_CtrleSingle.udiErrorID:=16#0;
			END_IF;
			(* init. variable *)
			xCalcAngleRefIndex:=FALSE;
		END_CASE;
	END_IF;

(* Send Axis Parameter *)
	IF xSendAxisParameter AND NOT(xBlockFBFunction) THEN
		CASE iStepSendPara OF
		(* control flag *)
		1:	udiFBErrorID:=0;
			(* Check first the usage of the correct parameter *)
			IF (iPtrAxisParameter = 1) AND (T_Axis.T_ParamFileObj[iPtrAxisParameter].udiIdxGroup = 0) THEN
				iStepSendPara:=91;
				RETURN;
			END_IF;
			udiIdxGroup:=T_Axis.T_ParamFileObj[iPtrAxisParameter].udiIdxGroup;
			udiIndexOffset:=T_Axis.T_ParamFileObj[iPtrAxisParameter].udiIndexOffset;
			udiLength:=T_Axis.T_ParamFileObj[iPtrAxisParameter].udiLength;
			lrReal:=T_Axis.T_ParamFileObj[iPtrAxisParameter].lrReal;
			SetObjectSDO:=TRUE;
			(* set next step  *)
			iStepSendPara:=iStepSendPara+1;
		2:	IF NOT(SetObjectSDO) THEN
				IF (T_Axis.T_ParamFileObj[iPtrAxisParameter + 1].udiIdxGroup <> 0) THEN
					(* next parameter *)
					iPtrAxisParameter:=iPtrAxisParameter+1;
					(* set next step  *)
					iStepSendPara:=1;
				ELSE
					(* set flag end function *)
					iStepSendPara:=99;
				END_IF;
			END_IF;
		(* Wrong paramter for this function *)
		91:	udiFBErrorID:=16#F20E;	(* Wrong Parameter for Function: Send Axis Parameter *)
			(* last step *)
			iStepSendPara:=99;
		(* init. done *)
		99:	IF (udiFBErrorID <> 0) THEN
				xFBErrorActive:=TRUE;
			END_IF;
			IF NOT(xFBErrorActive) THEN
				T_Axis.T_CtrleSingle.xDone:=TRUE;
				T_Axis.T_CtrleSingle.xErr:= FALSE;
				T_Axis.T_CtrleSingle.udiErrorID:=16#0;
			END_IF;
			(* init. variable *)
			xSendAxisParameter:=FALSE;
		END_CASE
	END_IF;

(* Send parameter to axis *)
	IF xSendPDOMappingPara AND NOT(xBlockFBFunction) THEN
		CASE iStepSendPara OF
		(* control flag *)
		1:	udiFBErrorID:=0;
			(* Check first the usage of the correct parameter *)
			IF (iPtrAxisParameter = 1) AND (T_Axis.T_ParamFileObj[iPtrAxisParameter].udiIdxGroup = 0) THEN
				iStepSendPara:=91;
				RETURN;
			END_IF;
			udiIdxGroup:=T_Axis.T_ParamFileObj[iPtrAxisParameter].udiIdxGroup;
			udiIndexOffset:=T_Axis.T_ParamFileObj[iPtrAxisParameter].udiIndexOffset;
			udiLength:=T_Axis.T_ParamFileObj[iPtrAxisParameter].udiLength;
			lrReal:=T_Axis.T_ParamFileObj[iPtrAxisParameter].lrReal;
			SetObjectSDO:=TRUE;
			(* set next step  *)
			iStepSendPara:=iStepSendPara+1;
		2:	IF NOT(SetObjectSDO) THEN
				IF (T_Axis.T_ParamFileObj[iPtrAxisParameter + 1].udiIdxGroup <> 0) THEN
					(* next parameter *)
					iPtrAxisParameter:=iPtrAxisParameter+1;
					(* set next step  *)
					iStepSendPara:=1;
				ELSE
					(* set flag end function *)
					iStepSendPara:=99;
				END_IF;
			END_IF;
		(* Wrong paramter for this function *)
		91:	udiFBErrorID:=16#F20F;	(* Wrong Parameter for Function: Send PDOMapping Parameter *)
			(* last step *)
			iStepSendPara:=99;
		(* init. done *)
		99:	IF (udiFBErrorID <> 0) THEN
				xFBErrorActive:=TRUE;
			END_IF;
			IF NOT(xFBErrorActive) THEN
				T_Axis.T_CtrleSingle.xDone:=TRUE;
				T_Axis.T_CtrleSingle.xErr:= FALSE;
				T_Axis.T_CtrleSingle.udiErrorID:=16#0;
			END_IF;
			(* init. variable *)
			xSendPDOMappingPara:=FALSE;
		END_CASE
	END_IF

(* Switch Master/Slave *)
	IF xMasterSlave AND NOT(xBlockFBFunction) THEN
		CASE iStepMasterSlave OF
		1:	udiFBErrorID:=0;
			(* Check first the usage of the correct parameter *)
			IF ((T_Axis.T_CtrleSingle.lrGearFactor = 0) OR (T_Axis.T_CtrleSingle.lrGearDivider = 0)) AND (siOpMode <> -4) THEN
				iStepMasterSlave:=91;
				RETURN;
			END_IF;
			udiIdxGroup:=16#6040;	(* Controlword *)
			udiIndexOffset:=16#0;
			udiLength:=16#2;
			lrReal:=16#F;
			SetObjectSDO:=TRUE;
			iStepMasterSlave:=iStepMasterSlave+1;
		2:	IF NOT(SetObjectSDO) THEN
				udiIdxGroup:=16#2509;	(* Mapping of the speed *)
				udiIndexOffset:=16#2;
				udiLength:=16#4;
				IF (siOpMode <> -4) THEN
					lrReal:=16#60FF0020;
				ELSE
					lrReal:=16#0;
				END_IF;
				SetObjectSDO:=TRUE;
				iStepMasterSlave:=iStepMasterSlave+1;
			END_IF;
		3:	IF NOT(SetObjectSDO) THEN
				IF (siOpMode <> -4) THEN
					udiIdxGroup:=16#2509;	(* Gear Factor *)
					udiIndexOffset:=16#3;
					udiLength:=16#2;
					lrReal:=T_Axis.T_CtrleSingle.lrGearFactor;
					SetObjectSDO:=TRUE;
				END_IF;
				iStepMasterSlave:=iStepMasterSlave+1;
			END_IF;
		4:	IF NOT(SetObjectSDO) THEN
				IF (siOpMode <> -4) THEN
					udiIdxGroup:=16#2509;	(* Gear Divider *)
					udiIndexOffset:=16#4;
					udiLength:=16#2;
					lrReal:=T_Axis.T_CtrleSingle.lrGearDivider;
					SetObjectSDO:=TRUE;
				END_IF;
				iStepMasterSlave:=iStepMasterSlave+1;
			END_IF;
		5:	IF NOT(SetObjectSDO) THEN
				udiIdxGroup:=16#2509;	(* Modus *)
				udiIndexOffset:=16#5;
				udiLength:=16#2;
				IF (siOpMode <> -4) THEN
					lrReal:=2;			(* Master/Slave *)
				ELSE
					lrReal:=0;			(* Master *)
				END_IF;
				SetObjectSDO:=TRUE;
				iStepMasterSlave:=iStepMasterSlave+1;
			END_IF;
		6:	IF NOT(SetObjectSDO) THEN
				udiIdxGroup:=16#6060;	(* mode of operation *)
				udiIndexOffset:=16#0;
				udiLength:=16#1;
				IF (siOpMode <> -4) THEN
					lrReal:=-4;
				ELSE
					lrReal:=1;
				END_IF;
				SetObjectSDO:=TRUE;
				iStepMasterSlave:=iStepMasterSlave+1;
			END_IF;
		7:	IF NOT(SetObjectSDO) AND ((UINT_TO_WORD(uiStatusWord) AND 16#4037) = 16#4037) THEN
				iStepMasterSlave:=99;
			END_IF;
		(* Wrong paramter for this function *)
		91:	udiFBErrorID:=16#F210;	(* Wrong Parameter for Function: Master/Slave *)
			(* last step *)
			iStepMasterSlave:=99;
		(* init. done *)
		99:	IF (udiFBErrorID <> 0) THEN
				xFBErrorActive:=TRUE;
			END_IF;
			IF NOT(xFBErrorActive) THEN
				T_Axis.T_CtrleSingle.xDone:=TRUE;
				T_Axis.T_CtrleSingle.xErr:= FALSE;
				T_Axis.T_CtrleSingle.udiErrorID:=16#0;
			END_IF;
			(* init. variable *)
			xMasterSlave:=FALSE;
		END_CASE;
	END_IF;

(* Save Parameter of Servo Drive *)
	IF xSaveParaEcoDrive AND NOT(xBlockFBFunction) THEN
		CASE iStepSaveParaEcoDrive OF
		1:	IF NOT(SetObjectSDO) THEN
				udiIdxGroup:=16#1010;	(* Save Objekt *)
				udiIndexOffset:=16#1;
				udiLength:=16#4;
				lrReal:=16#65766173;	(* Save all Ecostep Parameter *)
				SetObjectSDO:=TRUE;
				iStepSaveParaEcoDrive:=iStepSaveParaEcoDrive+1;
			END_IF;
		2:	IF NOT(SetObjectSDO) THEN
				T_Axis.T_CtrleSingle.xDone:=TRUE;
				T_Axis.T_CtrleSingle.xErr:= FALSE;
				T_Axis.T_CtrleSingle.udiErrorID:=0;
				(* init. variable *)
				xSaveParaEcoDrive:=FALSE;
			END_IF;
		END_CASE;
	END_IF;

(* Get Software Version EcoStep *)
	IF xGetSoftwareVersion AND NOT(xBlockFBFunction) THEN
		CASE iStepGetSoftwareVersion OF
		1:	IF NOT(GetObjectSDO) THEN
				udiIdxGroup:=16#2FE0;		(* Software version *)
				udiIndexOffset:=16#1;
				udiLength:=16#4;
				GetObjectSDO:=TRUE;
				iStepGetSoftwareVersion:=iStepGetSoftwareVersion + 1;
			END_IF;
		2:	IF NOT(GetObjectSDO) THEN
				T_Axis.T_SoftwareDetails.lrSoftwareVersion:=lrReal;
				udiIdxGroup:=16#2FE0;		(* Build version *)
				udiIndexOffset:=16#2;
				udiLength:=16#4;
				GetObjectSDO:=TRUE;
				iStepGetSoftwareVersion:=iStepGetSoftwareVersion + 1;
			END_IF;
		3:	IF NOT(GetObjectSDO) THEN
				T_Axis.T_SoftwareDetails.lrBuildVersion:=lrReal;
				udiIdxGroup:=16#2FE0;		(* Software date code *)
				udiIndexOffset:=16#3;
				udiLength:=16#4;
				GetObjectSDO:=TRUE;
				iStepGetSoftwareVersion:=iStepGetSoftwareVersion + 1;
			END_IF;
		4:	IF NOT(GetObjectSDO) THEN
				T_Axis.T_SoftwareDetails.lrDateCode:=lrReal;
				sCopyDateCode:=LREAL_TO_STRING(lrReal);
				sTmpDateCode:=MID(sCopyDateCode,2,7);	(* Get Day *)
				sTmpDateCode:=CONCAT(sTmpDateCode,'.');
				sTmpDateCode:=CONCAT(sTmpDateCode,MID(sCopyDateCode,2,5));	(* Get Month *)
				sTmpDateCode:=CONCAT(sTmpDateCode,'.');
				sTmpDateCode:=CONCAT(sTmpDateCode,MID(sCopyDateCode,4,1));	(* Get Year *)
				T_Axis.T_SoftwareDetails.sDateCode:=sTmpDateCode;
				T_Axis.T_CtrleSingle.xDone:=TRUE;
				T_Axis.T_CtrleSingle.xErr:= FALSE;
				T_Axis.T_CtrleSingle.udiErrorID:=0;
				(* init. variable *)
				xGetSoftwareVersion:=FALSE;
			END_IF;
		END_CASE;
	END_IF;

(* Set Software limit switch *)
	IF xSetSWLimitSwitch AND NOT(xBlockFBFunction) THEN
		CASE iStepSetSWLimitSwitch OF
		1:	IF NOT(SetObjectSDO) THEN
				udiIdxGroup:=16#607D;	(* Object for the SW Limit switch *)
				udiIndexOffset:=16#1;	(* Subindex for the neg end switch *)
				udiLength:=16#4;
				IF (T_Axis.T_Config_Gen.iTyp <> 5) THEN
					lrReal:=T_Axis.T_CtrleSingle.lrSWNegLimitSwitch * T_Axis.T_CtrleSingle.lrScaleFactor;
				ELSE
					lrReal:=T_Axis.T_CtrleSingle.lrSWNegLimitSwitch * T_Axis.T_CtrleSingle.lrScaleFactor * rPrismaFactor;
				END_IF;
				SetObjectSDO:=TRUE;
				iStepSetSWLimitSwitch:=iStepSetSWLimitSwitch+1;
			END_IF;
		2:	IF NOT(SetObjectSDO) THEN
				udiIdxGroup:=16#607D;	(* Object for the SW Limit switch *)
				udiIndexOffset:=16#2;	(* Subindex for the pos end switch *)
				udiLength:=16#4;
				IF (T_Axis.T_Config_Gen.iTyp <> 5) THEN
					lrReal:=T_Axis.T_CtrleSingle.lrSWPosLimitSwitch * T_Axis.T_CtrleSingle.lrScaleFactor;
				ELSE
					lrReal:=T_Axis.T_CtrleSingle.lrSWPosLimitSwitch * T_Axis.T_CtrleSingle.lrScaleFactor * rPrismaFactor;
				END_IF;
				SetObjectSDO:=TRUE;
				iStepSetSWLimitSwitch:=iStepSetSWLimitSwitch+1;
			END_IF;
		3:	IF NOT(SetObjectSDO) THEN
				T_Axis.T_CtrleSingle.xDone:=TRUE;
				T_Axis.T_CtrleSingle.xErr:= FALSE;
				T_Axis.T_CtrleSingle.udiErrorID:=0;
				(* init. variable *)
				xSetSWLimitSwitch:=FALSE;
			END_IF;
		END_CASE;
	END_IF;

(* Reset Software limit switch *)
	IF xResetSWLimitSwitch AND NOT(xBlockFBFunction) THEN
		CASE iStepResetSWLimitSwitch OF
		1:	IF NOT(SetObjectSDO) THEN
				udiIdxGroup:=16#607D;	(* Object for the SW Limit switch *)
				udiIndexOffset:=16#1;	(* Subindex for the neg end switch *)
				udiLength:=16#4;
				lrReal:=0;
				SetObjectSDO:=TRUE;
				iStepResetSWLimitSwitch:=iStepResetSWLimitSwitch+1;
			END_IF;
		2:	IF NOT(SetObjectSDO) THEN
				udiIdxGroup:=16#607D;	(* Object for the SW Limit switch *)
				udiIndexOffset:=16#2;	(* Subindex for the pos end switch *)
				udiLength:=16#4;
				lrReal:=0;
				SetObjectSDO:=TRUE;
				iStepResetSWLimitSwitch:=iStepResetSWLimitSwitch+1;
			END_IF;
		3:	IF NOT(SetObjectSDO) THEN
				T_Axis.T_CtrleSingle.xDone:=TRUE;
				T_Axis.T_CtrleSingle.xErr:= FALSE;
				T_Axis.T_CtrleSingle.udiErrorID:=0;
				(* init. variable *)
				xResetSWLimitSwitch:=FALSE;
			END_IF;
		END_CASE;
	END_IF;

(* send set SDO Object *)
	IF SetObjectSDO THEN
		IF (udiIdxGroup = 16#6040) THEN
			lrSettledControlword:=lrReal;
		END_IF;
		FBSetObjectSDO(		ADSNetId:=T_Axis.T_Config_Gen.sAmsNetId,
							NodeId:=UDINT_TO_INT(T_Axis.T_Config_Gen.udiNodeId),
							Write:=TRUE,
							ObjectIndex:=UDINT_TO_UINT(udiIdxGroup),
							ObjectSubIndex:=UDINT_TO_USINT(udiIndexOffset),
							LEN:=UDINT_TO_USINT(udiLength),
							Data:=LREAL_TO_UDINT(lrReal));
		IF FBSetObjectSDO.Done AND NOT(FBSetObjectSDO.ERR) THEN
			FBSetObjectSDO(Write:=FALSE);
			SetObjectSDO:=FALSE;
		END_IF;
		IF FBSetObjectSDO.ERR THEN
			xADSErrorActive:=TRUE;
			udiADSErrorID:=FBSetObjectSDO.ErrNo;
			FBSetObjectSDO(Write:=FALSE);
			SetObjectSDO:=FALSE;
		END_IF;
	ELSE
		FBSetObjectSDO(Write:=FALSE);
	END_IF;

